LIN {X 0,Y 523.952,Z 123.214,A -85,B 0,C 180,E1 -4834.581,E2 -4834.581} C_VEL
LIN {X 0,Y 523.913,Z 123.226,A -85,B 0,C 180,E1 -4837.106,E2 -4837.106} C_VEL
LIN {X 0,Y 523.982,Z 123.211,A -85,B 0,C 180,E1 -4839.866,E2 -4839.866} C_VEL
LIN {X 0,Y 523.946,Z 123.22,A -85,B 0,C 180,E1 -4842.836,E2 -4842.836} C_VEL
LIN {X 0,Y 523.977,Z 123.217,A -85,B 0,C 180,E1 -4845.235,E2 -4845.235} C_VEL
LIN {X 0,Y 524.016,Z 123.21,A -85,B 0,C 180,E1 -4848.394,E2 -4848.394} C_VEL
LIN {X 0,Y 523.99,Z 123.212,A -85,B 0,C 180,E1 -4851.515,E2 -4851.515} C_VEL
LIN {X 0,Y 524.08,Z 123.208,A -85,B 0,C 180,E1 -4854.613,E2 -4854.613} C_VEL
LIN {X 0,Y 524.112,Z 123.197,A -85,B 0,C 180,E1 -4857.694,E2 -4857.694} C_VEL
LIN {X 0,Y 524.121,Z 123.2,A -85,B 0,C 180,E1 -4860.768,E2 -4860.768} C_VEL
LIN {X 0,Y 524.032,Z 123.209,A -85,B 0,C 180,E1 -4863.075,E2 -4863.075} C_VEL
LIN {X 0,Y 524.035,Z 123.213,A -85,B 0,C 180,E1 -4866.159,E2 -4866.159} C_VEL
LIN {X 0,Y 524.063,Z 123.317,A -85,B 0,C 180,E1 -4866.954,E2 -4866.954} C_VEL
LIN {X 0,Y 524.293,Z 129.392,A -85,B 0,C 180,E1 -4868.091,E2 -4868.091} C_VEL
LIN {X 0,Y 524.223,Z 139.02,A -85,B 0,C 180,E1 -4869.915,E2 -4869.915} C_VEL
LIN {X 0,Y 525.974,Z 147.912,A -85,B 0,C 180,E1 -4870.1,E2 -4870.1} C_VEL
LIN {X 0,Y 525.464,Z 245.35,A -85,B 0,C 180,E1 -4871.5,E2 -4871.5} C_VEL
LIN {X 0,Y 525.299,Z 258.517,A -85,B 0,C 180,E1 -4871.84,E2 -4871.84} C_VEL
LIN {X 0,Y 525.121,Z 270.833,A -85,B 0,C 180,E1 -4872.311,E2 -4872.311} C_VEL
LIN {X 0,Y 524.861,Z 283.293,A -85,B 0,C 180,E1 -4872.961,E2 -4872.961} C_VEL
LIN {X 0,Y 524.562,Z 295.002,A -85,B 0,C 180,E1 -4873.757,E2 -4873.757} C_VEL
LIN {X 0,Y 524.314,Z 305.505,A -85,B 0,C 180,E1 -4874.655,E2 -4874.655} C_VEL
LIN {X 0,Y 524.119,Z 314.056,A -85,B 0,C 180,E1 -4875.556,E2 -4875.556} C_VEL
LIN {X 0,Y 523.845,Z 323.352,A -85,B 0,C 180,E1 -4876.765,E2 -4876.765} C_VEL
LIN {X 0,Y 523.686,Z 330.798,A -85,B 0,C 180,E1 -4877.979,E2 -4877.979} C_VEL
LIN {X 0,Y 523.617,Z 336.668,A -85,B 0,C 180,E1 -4879.198,E2 -4879.198} C_VEL
LIN {X 0,Y 523.481,Z 341.276,A -85,B 0,C 180,E1 -4880.43,E2 -4880.43} C_VEL
LIN {X 0,Y 523.428,Z 343.689,A -85,B 0,C 180,E1 -4881.255,E2 -4881.255} C_VEL
LIN {X 0,Y 523.372,Z 345.621,A -85,B 0,C 180,E1 -4882.096,E2 -4882.096} C_VEL
LIN {X 0,Y 523.31,Z 347.024,A -85,B 0,C 180,E1 -4882.921,E2 -4882.921} C_VEL
LIN {X 0,Y 523.288,Z 348.184,A -85,B 0,C 180,E1 -4884.038,E2 -4884.038} C_VEL
LIN {X 0,Y 523.308,Z 348.449,A -85,B 0,C 180,E1 -4885.452,E2 -4885.452} C_VEL
LIN {X 0,Y 523.314,Z 347.985,A -85,B 0,C 180,E1 -4886.307,E2 -4886.307} C_VEL
LIN {X 0,Y 523.362,Z 346.319,A -85,B 0,C 180,E1 -4887.589,E2 -4887.589} C_VEL
LIN {X 0,Y 523.419,Z 343.417,A -85,B 0,C 180,E1 -4888.906,E2 -4888.906} C_VEL
LIN {X 0,Y 523.476,Z 339.204,A -85,B 0,C 180,E1 -4890.229,E2 -4890.229} C_VEL
LIN {X 0,Y 523.489,Z 338.508,A -85,B 0,C 180,E1 -4890.408,E2 -4890.408} C_VEL
LIN {X 0,Y 522.873,Z 336.184,A -85,B 0,C 180,E1 -4890.998,E2 -4890.998} C_VEL
LIN {X 0,Y 520.085,Z 331.973,A -85,B 0,C 180,E1 -4891.94,E2 -4891.94} C_VEL
LIN {X 0,Y 517.343,Z 327.2,A -85,B 0,C 180,E1 -4892.853,E2 -4892.853} C_VEL
LIN {X 0,Y 516.804,Z 323.835,A -85,B 0,C 180,E1 -4893.39,E2 -4893.39} C_VEL
LIN {X 0,Y 517.078,Z 314.887,A -85,B 0,C 180,E1 -4894.578,E2 -4894.578} C_VEL
LIN {X 0,Y 517.334,Z 305.085,A -85,B 0,C 180,E1 -4895.625,E2 -4895.625} C_VEL
LIN {X 0,Y 517.652,Z 294.078,A -85,B 0,C 180,E1 -4896.561,E2 -4896.561} C_VEL
LIN {X 0,Y 517.921,Z 283.602,A -85,B 0,C 180,E1 -4897.276,E2 -4897.276} C_VEL
LIN {X 0,Y 518.173,Z 272.168,A -85,B 0,C 180,E1 -4897.893,E2 -4897.893} C_VEL
LIN {X 0,Y 518.298,Z 259.428,A -85,B 0,C 180,E1 -4898.402,E2 -4898.402} C_VEL
LIN {X 0,Y 518.52,Z 246.192,A -85,B 0,C 180,E1 -4898.757,E2 -4898.757} C_VEL
LIN {X 0,Y 519.003,Z 147.832,A -85,B 0,C 180,E1 -4900.198,E2 -4900.198} C_VEL
LIN {X 0,Y 517.241,Z 138.787,A -85,B 0,C 180,E1 -4900.405,E2 -4900.405} C_VEL
LIN {X 0,Y 517.335,Z 126.807,A -85,B 0,C 180,E1 -4902.811,E2 -4902.811} C_VEL
LIN {X 0,Y 516.956,Z 124.094,A -85,B 0,C 180,E1 -4903.426,E2 -4903.426} C_VEL
LIN {X 0,Y 516.883,Z 124.101,A -85,B 0,C 180,E1 -4906.107,E2 -4906.107} C_VEL
LIN {X 0,Y 516.915,Z 124.092,A -85,B 0,C 180,E1 -4908.398,E2 -4908.398} C_VEL
LIN {X 0,Y 516.88,Z 124.099,A -85,B 0,C 180,E1 -4911.284,E2 -4911.284} C_VEL
LIN {X 0,Y 516.87,Z 124.098,A -85,B 0,C 180,E1 -4914.219,E2 -4914.219} C_VEL
LIN {X 0,Y 516.88,Z 124.098,A -85,B 0,C 180,E1 -4917.052,E2 -4917.052} C_VEL
LIN {X 0,Y 516.886,Z 124.098,A -85,B 0,C 180,E1 -4919.796,E2 -4919.796} C_VEL
LIN {X 0,Y 516.925,Z 124.089,A -85,B 0,C 180,E1 -4922.467,E2 -4922.467} C_VEL
LIN {X 0,Y 516.908,Z 124.096,A -85,B 0,C 180,E1 -4925.071,E2 -4925.071} C_VEL
LIN {X 0,Y 516.885,Z 124.095,A -85,B 0,C 180,E1 -4928.462,E2 -4928.462} C_VEL
LIN {X 0,Y 516.899,Z 124.098,A -85,B 0,C 180,E1 -4930.954,E2 -4930.954} C_VEL
LIN {X 0,Y 516.907,Z 124.097,A -85,B 0,C 180,E1 -4933.41,E2 -4933.41} C_VEL
LIN {X 0,Y 516.894,Z 124.094,A -85,B 0,C 180,E1 -4935.833,E2 -4935.833} C_VEL
LIN {X 0,Y 516.965,Z 124.085,A -85,B 0,C 180,E1 -4938.233,E2 -4938.233} C_VEL
LIN {X 0,Y 516.967,Z 124.088,A -85,B 0,C 180,E1 -4941.399,E2 -4941.399} C_VEL
LIN {X 0,Y 517.001,Z 124.08,A -85,B 0,C 180,E1 -4943.756,E2 -4943.756} C_VEL
LIN {X 0,Y 517.012,Z 124.088,A -85,B 0,C 180,E1 -4946.883,E2 -4946.883} C_VEL
LIN {X 0,Y 517.085,Z 124.07,A -85,B 0,C 180,E1 -4950,E2 -4950} C_VEL
LIN {X 0,Y 517.01,Z 124.083,A -85,B 0,C 180,E1 -4953.117,E2 -4953.117} C_VEL
LIN {X 0,Y 517.002,Z 124.083,A -85,B 0,C 180,E1 -4956.243,E2 -4956.243} C_VEL
LIN {X 0,Y 516.952,Z 124.087,A -85,B 0,C 180,E1 -4959.389,E2 -4959.389} C_VEL
LIN {X 0,Y 516.951,Z 124.087,A -85,B 0,C 180,E1 -4961.807,E2 -4961.807} C_VEL
LIN {X 0,Y 516.945,Z 124.088,A -85,B 0,C 180,E1 -4965.147,E2 -4965.147} C_VEL
LIN {X 0,Y 516.923,Z 124.096,A -85,B 0,C 180,E1 -4968.222,E2 -4968.222} C_VEL
LIN {X 0,Y 516.91,Z 124.095,A -85,B 0,C 180,E1 -4970.701,E2 -4970.701} C_VEL
LIN {X 0,Y 516.888,Z 124.1,A -85,B 0,C 180,E1 -4974.073,E2 -4974.073} C_VEL
LIN {X 0,Y 516.922,Z 124.093,A -85,B 0,C 180,E1 -4976.658,E2 -4976.658} C_VEL
LIN {X 0,Y 516.917,Z 124.092,A -85,B 0,C 180,E1 -4979.525,E2 -4979.525} C_VEL
LIN {X 0,Y 516.898,Z 124.096,A -85,B 0,C 180,E1 -4982.544,E2 -4982.544} C_VEL
LIN {X 0,Y 516.877,Z 124.096,A -85,B 0,C 180,E1 -4985.332,E2 -4985.332} C_VEL
LIN {X 0,Y 516.879,Z 124.104,A -85,B 0,C 180,E1 -4987.943,E2 -4987.943} C_VEL
LIN {X 0,Y 516.883,Z 124.095,A -85,B 0,C 180,E1 -4990.741,E2 -4990.741} C_VEL
LIN {X 0,Y 516.902,Z 124.092,A -85,B 0,C 180,E1 -4992.829,E2 -4992.829} C_VEL
LIN {X 0,Y 516.919,Z 124.09,A -85,B 0,C 180,E1 -4995.01,E2 -4995.01} C_VEL
LIN {X 0,Y 516.92,Z 124.091,A -85,B 0,C 180,E1 -4998.398,E2 -4998.398} C_VEL
LIN {X 0,Y 516.884,Z 124.098,A -85,B 0,C 180,E1 -5001.285,E2 -5001.285} C_VEL
LIN {X 0,Y 516.868,Z 124.098,A -85,B 0,C 180,E1 -5004.22,E2 -5004.22} C_VEL
LIN {X 0,Y 516.894,Z 124.095,A -85,B 0,C 180,E1 -5007.053,E2 -5007.053} C_VEL
LIN {X 0,Y 516.889,Z 124.099,A -85,B 0,C 180,E1 -5009.796,E2 -5009.796} C_VEL
LIN {X 0,Y 516.925,Z 124.089,A -85,B 0,C 180,E1 -5012.468,E2 -5012.468} C_VEL
LIN {X 0,Y 516.906,Z 124.096,A -85,B 0,C 180,E1 -5015.072,E2 -5015.072} C_VEL
LIN {X 0,Y 516.883,Z 124.095,A -85,B 0,C 180,E1 -5018.462,E2 -5018.462} C_VEL
LIN {X 0,Y 516.901,Z 124.097,A -85,B 0,C 180,E1 -5020.955,E2 -5020.955} C_VEL
LIN {X 0,Y 516.911,Z 124.098,A -85,B 0,C 180,E1 -5023.41,E2 -5023.41} C_VEL
LIN {X 0,Y 516.892,Z 124.095,A -85,B 0,C 180,E1 -5025.834,E2 -5025.834} C_VEL
LIN {X 0,Y 516.963,Z 124.085,A -85,B 0,C 180,E1 -5028.234,E2 -5028.234} C_VEL
LIN {X 0,Y 516.966,Z 124.088,A -85,B 0,C 180,E1 -5031.4,E2 -5031.4} C_VEL
LIN {X 0,Y 517.001,Z 124.081,A -85,B 0,C 180,E1 -5033.757,E2 -5033.757} C_VEL
LIN {X 0,Y 517.011,Z 124.087,A -85,B 0,C 180,E1 -5036.883,E2 -5036.883} C_VEL
LIN {X 0,Y 517.084,Z 124.07,A -85,B 0,C 180,E1 -5040,E2 -5040} C_VEL
LIN {X 0,Y 517.01,Z 124.083,A -85,B 0,C 180,E1 -5043.117,E2 -5043.117} C_VEL
LIN {X 0,Y 517.014,Z 124.081,A -85,B 0,C 180,E1 -5046.243,E2 -5046.243} C_VEL
LIN {X 0,Y 516.953,Z 124.087,A -85,B 0,C 180,E1 -5049.39,E2 -5049.39} C_VEL
LIN {X 0,Y 516.951,Z 124.087,A -85,B 0,C 180,E1 -5051.808,E2 -5051.808} C_VEL
LIN {X 0,Y 516.946,Z 124.088,A -85,B 0,C 180,E1 -5055.148,E2 -5055.148} C_VEL
LIN {X 0,Y 516.924,Z 124.095,A -85,B 0,C 180,E1 -5058.223,E2 -5058.223} C_VEL
LIN {X 0,Y 516.912,Z 124.096,A -85,B 0,C 180,E1 -5060.702,E2 -5060.702} C_VEL
LIN {X 0,Y 516.89,Z 124.099,A -85,B 0,C 180,E1 -5064.073,E2 -5064.073} C_VEL
LIN {X 0,Y 516.924,Z 124.093,A -85,B 0,C 180,E1 -5066.658,E2 -5066.658} C_VEL
LIN {X 0,Y 516.91,Z 124.092,A -85,B 0,C 180,E1 -5069.524,E2 -5069.524} C_VEL
LIN {X 0,Y 516.895,Z 124.097,A -85,B 0,C 180,E1 -5072.544,E2 -5072.544} C_VEL
LIN {X 0,Y 516.865,Z 124.097,A -85,B 0,C 180,E1 -5075.33,E2 -5075.33} C_VEL
LIN {X 0,Y 516.881,Z 124.102,A -85,B 0,C 180,E1 -5077.944,E2 -5077.944} C_VEL
LIN {X 0,Y 516.895,Z 124.094,A -85,B 0,C 180,E1 -5080.741,E2 -5080.741} C_VEL
LIN {X 0,Y 516.883,Z 124.104,A -85,B 0,C 180,E1 -5083.904,E2 -5083.904} C_VEL
LIN {X 0,Y 516.883,Z 124.1,A -85,B 0,C 180,E1 -5086.107,E2 -5086.107} C_VEL
LIN {X 0,Y 516.917,Z 124.092,A -85,B 0,C 180,E1 -5088.399,E2 -5088.399} C_VEL
LIN {X 0,Y 516.884,Z 124.097,A -85,B 0,C 180,E1 -5091.285,E2 -5091.285} C_VEL
LIN {X 0,Y 516.872,Z 124.098,A -85,B 0,C 180,E1 -5094.22,E2 -5094.22} C_VEL
LIN {X 0,Y 516.896,Z 124.095,A -85,B 0,C 180,E1 -5097.053,E2 -5097.053} C_VEL
LIN {X 0,Y 516.893,Z 124.1,A -85,B 0,C 180,E1 -5099.797,E2 -5099.797} C_VEL
LIN {X 0,Y 516.928,Z 124.091,A -85,B 0,C 180,E1 -5102.468,E2 -5102.468} C_VEL
LIN {X 0,Y 516.957,Z 124.191,A -85,B 0,C 180,E1 -5104.402,E2 -5104.402} C_VEL
LIN {X 0,Y 518.636,Z 133.005,A -85,B 0,C 180,E1 -5105.836,E2 -5105.836} C_VEL
LIN {X 0,Y 518.274,Z 148.017,A -85,B 0,C 180,E1 -5108.105,E2 -5108.105} C_VEL
LIN {X 0,Y 517.818,Z 167.379,A -85,B 0,C 180,E1 -5110.99,E2 -5110.99} C_VEL
LIN {X 0,Y 517.345,Z 186.704,A -85,B 0,C 180,E1 -5113.83,E2 -5113.83} C_VEL
LIN {X 0,Y 517.246,Z 192.193,A -85,B 0,C 180,E1 -5114.633,E2 -5114.633} C_VEL
LIN {X 0,Y 518.989,Z 205.615,A -85,B 0,C 180,E1 -5114.884,E2 -5114.884} C_VEL
LIN {X 0,Y 518.489,Z 301.678,A -85,B 0,C 180,E1 -5116.278,E2 -5116.278} C_VEL
LIN {X 0,Y 518.244,Z 314.629,A -85,B 0,C 180,E1 -5116.622,E2 -5116.622} C_VEL
LIN {X 0,Y 517.964,Z 327.229,A -85,B 0,C 180,E1 -5117.113,E2 -5117.113} C_VEL
LIN {X 0,Y 517.645,Z 339.245,A -85,B 0,C 180,E1 -5117.752,E2 -5117.752} C_VEL
LIN {X 0,Y 517.35,Z 350.788,A -85,B 0,C 180,E1 -5118.541,E2 -5118.541} C_VEL
LIN {X 0,Y 517.118,Z 361.192,A -85,B 0,C 180,E1 -5119.428,E2 -5119.428} C_VEL
LIN {X 0,Y 516.831,Z 370.527,A -85,B 0,C 180,E1 -5120.411,E2 -5120.411} C_VEL
LIN {X 0,Y 516.617,Z 379.595,A -85,B 0,C 180,E1 -5121.591,E2 -5121.591} C_VEL
LIN {X 0,Y 516.461,Z 386.898,A -85,B 0,C 180,E1 -5122.769,E2 -5122.769} C_VEL
LIN {X 0,Y 516.372,Z 391.826,A -85,B 0,C 180,E1 -5123.749,E2 -5123.749} C_VEL
LIN {X 0,Y 516.312,Z 396.613,A -85,B 0,C 180,E1 -5124.924,E2 -5124.924} C_VEL
LIN {X 0,Y 516.37,Z 400.275,A -85,B 0,C 180,E1 -5126.098,E2 -5126.098} C_VEL
LIN {X 0,Y 516.327,Z 402.159,A -85,B 0,C 180,E1 -5126.879,E2 -5126.879} C_VEL
LIN {X 0,Y 516.266,Z 403.569,A -85,B 0,C 180,E1 -5127.66,E2 -5127.66} C_VEL
LIN {X 0,Y 516.182,Z 405.179,A -85,B 0,C 180,E1 -5129.22,E2 -5129.22} C_VEL
LIN {X 0,Y 516.186,Z 405.391,A -85,B 0,C 180,E1 -5130,E2 -5130} C_VEL
LIN {X 0,Y 516.182,Z 405.165,A -85,B 0,C 180,E1 -5130.78,E2 -5130.78} C_VEL
LIN {X 0,Y 516.266,Z 403.524,A -85,B 0,C 180,E1 -5132.341,E2 -5132.341} C_VEL
LIN {X 0,Y 516.327,Z 402.097,A -85,B 0,C 180,E1 -5133.121,E2 -5133.121} C_VEL
LIN {X 0,Y 516.312,Z 399.099,A -85,B 0,C 180,E1 -5134.294,E2 -5134.294} C_VEL
LIN {X 0,Y 516.389,Z 395.048,A -85,B 0,C 180,E1 -5135.467,E2 -5135.467} C_VEL
LIN {X 0,Y 516.416,Z 388.803,A -85,B 0,C 180,E1 -5136.84,E2 -5136.84} C_VEL
LIN {X 0,Y 516.563,Z 381.996,A -85,B 0,C 180,E1 -5138.017,E2 -5138.017} C_VEL
LIN {X 0,Y 516.74,Z 373.54,A -85,B 0,C 180,E1 -5139.196,E2 -5139.196} C_VEL
LIN {X 0,Y 516.935,Z 364.836,A -85,B 0,C 180,E1 -5140.18,E2 -5140.18} C_VEL
LIN {X 0,Y 517.253,Z 354.109,A -85,B 0,C 180,E1 -5141.164,E2 -5141.164} C_VEL
LIN {X 0,Y 517.492,Z 342.601,A -85,B 0,C 180,E1 -5142.012,E2 -5142.012} C_VEL
LIN {X 0,Y 517.793,Z 330.687,A -85,B 0,C 180,E1 -5142.692,E2 -5142.692} C_VEL
LIN {X 0,Y 518.108,Z 318.162,A -85,B 0,C 180,E1 -5143.233,E2 -5143.233} C_VEL
LIN {X 0,Y 518.355,Z 305.212,A -85,B 0,C 180,E1 -5143.626,E2 -5143.626} C_VEL
LIN {X 0,Y 518.548,Z 289.822,A -85,B 0,C 180,E1 -5143.895,E2 -5143.895} C_VEL
LIN {X 0,Y 518.851,Z 203.924,A -85,B 0,C 180,E1 -5145.135,E2 -5145.135} C_VEL
LIN {X 0,Y 517.179,Z 191.339,A -85,B 0,C 180,E1 -5145.382,E2 -5145.382} C_VEL
LIN {X 0,Y 517.63,Z 168.939,A -85,B 0,C 180,E1 -5148.607,E2 -5148.607} C_VEL
LIN {X 0,Y 517.938,Z 149.08,A -85,B 0,C 180,E1 -5151.492,E2 -5151.492} C_VEL
LIN {X 0,Y 518.301,Z 132.004,A -85,B 0,C 180,E1 -5154.004,E2 -5154.004} C_VEL
LIN {X 0,Y 516.973,Z 124.09,A -85,B 0,C 180,E1 -5155.248,E2 -5155.248} C_VEL
LIN {X 0,Y 516.922,Z 124.102,A -85,B 0,C 180,E1 -5158.415,E2 -5158.415} C_VEL
LIN {X 0,Y 516.893,Z 124.098,A -85,B 0,C 180,E1 -5161.11,E2 -5161.11} C_VEL
LIN {X 0,Y 516.912,Z 124.098,A -85,B 0,C 180,E1 -5163.966,E2 -5163.966} C_VEL
LIN {X 0,Y 516.88,Z 124.098,A -85,B 0,C 180,E1 -5166.746,E2 -5166.746} C_VEL
LIN {X 0,Y 516.886,Z 124.101,A -85,B 0,C 180,E1 -5169.721,E2 -5169.721} C_VEL
LIN {X 0,Y 516.915,Z 124.098,A -85,B 0,C 180,E1 -5171.775,E2 -5171.775} C_VEL
LIN {X 0,Y 516.927,Z 124.091,A -85,B 0,C 180,E1 -5175.01,E2 -5175.01} C_VEL
LIN {X 0,Y 516.917,Z 124.091,A -85,B 0,C 180,E1 -5178.399,E2 -5178.399} C_VEL
LIN {X 0,Y 516.884,Z 124.097,A -85,B 0,C 180,E1 -5181.284,E2 -5181.284} C_VEL
LIN {X 0,Y 516.874,Z 124.097,A -85,B 0,C 180,E1 -5184.22,E2 -5184.22} C_VEL
LIN {X 0,Y 516.884,Z 124.096,A -85,B 0,C 180,E1 -5187.052,E2 -5187.052} C_VEL
LIN {X 0,Y 516.89,Z 124.098,A -85,B 0,C 180,E1 -5189.796,E2 -5189.796} C_VEL
LIN {X 0,Y 516.928,Z 124.09,A -85,B 0,C 180,E1 -5192.467,E2 -5192.467} C_VEL
LIN {X 0,Y 516.909,Z 124.096,A -85,B 0,C 180,E1 -5195.071,E2 -5195.071} C_VEL
LIN {X 0,Y 516.888,Z 124.096,A -85,B 0,C 180,E1 -5198.462,E2 -5198.462} C_VEL
LIN {X 0,Y 516.895,Z 124.1,A -85,B 0,C 180,E1 -5200.954,E2 -5200.954} C_VEL
LIN {X 0,Y 516.901,Z 124.096,A -85,B 0,C 180,E1 -5203.409,E2 -5203.409} C_VEL
LIN {X 0,Y 516.89,Z 124.095,A -85,B 0,C 180,E1 -5205.833,E2 -5205.833} C_VEL
LIN {X 0,Y 516.953,Z 124.094,A -85,B 0,C 180,E1 -5209.028,E2 -5209.028} C_VEL
LIN {X 0,Y 516.965,Z 124.089,A -85,B 0,C 180,E1 -5212.186,E2 -5212.186} C_VEL
LIN {X 0,Y 517.027,Z 124.086,A -85,B 0,C 180,E1 -5214.54,E2 -5214.54} C_VEL
LIN {X 0,Y 517.083,Z 124.073,A -85,B 0,C 180,E1 -5217.663,E2 -5217.663} C_VEL
LIN {X 0,Y 517.091,Z 124.076,A -85,B 0,C 180,E1 -5220.778,E2 -5220.778} C_VEL
LIN {X 0,Y 516.974,Z 124.088,A -85,B 0,C 180,E1 -5223.117,E2 -5223.117} C_VEL
LIN {X 0,Y 517.001,Z 124.09,A -85,B 0,C 180,E1 -5226.243,E2 -5226.243} C_VEL
LIN {X 0,Y 516.988,Z 124.135,A -85,B 0,C 180,E1 -5226.817,E2 -5226.817} C_VEL
LIN {X 0,Y 517.351,Z 129.359,A -85,B 0,C 180,E1 -5227.807,E2 -5227.807} C_VEL
LIN {X 0,Y 517.256,Z 139.386,A -85,B 0,C 180,E1 -5229.704,E2 -5229.704} C_VEL
LIN {X 0,Y 519.133,Z 149.215,A -85,B 0,C 180,E1 -5229.915,E2 -5229.915} C_VEL
LIN {X 0,Y 518.556,Z 246.037,A -85,B 0,C 180,E1 -5231.333,E2 -5231.333} C_VEL
LIN {X 0,Y 518.384,Z 259.286,A -85,B 0,C 180,E1 -5231.684,E2 -5231.684} C_VEL
LIN {X 0,Y 518.205,Z 272.025,A -85,B 0,C 180,E1 -5232.185,E2 -5232.185} C_VEL
LIN {X 0,Y 517.906,Z 284.191,A -85,B 0,C 180,E1 -5232.839,E2 -5232.839} C_VEL
LIN {X 0,Y 517.6,Z 295.81,A -85,B 0,C 180,E1 -5233.645,E2 -5233.645} C_VEL
LIN {X 0,Y 517.311,Z 306.237,A -85,B 0,C 180,E1 -5234.556,E2 -5234.556} C_VEL
LIN {X 0,Y 517.063,Z 315.866,A -85,B 0,C 180,E1 -5235.607,E2 -5235.607} C_VEL
LIN {X 0,Y 516.81,Z 324.684,A -85,B 0,C 180,E1 -5236.796,E2 -5236.796} C_VEL
LIN {X 0,Y 516.638,Z 331.539,A -85,B 0,C 180,E1 -5237.956,E2 -5237.956} C_VEL
LIN {X 0,Y 516.552,Z 336.797,A -85,B 0,C 180,E1 -5239.058,E2 -5239.058} C_VEL
LIN {X 0,Y 516.431,Z 340.847,A -85,B 0,C 180,E1 -5240.114,E2 -5240.114} C_VEL
LIN {X 0,Y 516.331,Z 344.945,A -85,B 0,C 180,E1 -5241.562,E2 -5241.562} C_VEL
LIN {X 0,Y 516.262,Z 346.658,A -85,B 0,C 180,E1 -5242.406,E2 -5242.406} C_VEL
LIN {X 0,Y 516.205,Z 347.893,A -85,B 0,C 180,E1 -5243.255,E2 -5243.255} C_VEL
LIN {X 0,Y 516.19,Z 348.67,A -85,B 0,C 180,E1 -5244.186,E2 -5244.186} C_VEL
LIN {X 0,Y 516.185,Z 348.913,A -85,B 0,C 180,E1 -5244.965,E2 -5244.965} C_VEL
LIN {X 0,Y 516.248,Z 348.561,A -85,B 0,C 180,E1 -5246.038,E2 -5246.038} C_VEL
LIN {X 0,Y 516.274,Z 346.801,A -85,B 0,C 180,E1 -5247.57,E2 -5247.57} C_VEL
LIN {X 0,Y 516.334,Z 343.965,A -85,B 0,C 180,E1 -5248.894,E2 -5248.894} C_VEL
LIN {X 0,Y 516.406,Z 339.798,A -85,B 0,C 180,E1 -5250.235,E2 -5250.235} C_VEL
LIN {X 0,Y 516.577,Z 334.142,A -85,B 0,C 180,E1 -5251.586,E2 -5251.586} C_VEL
LIN {X 0,Y 516.746,Z 328.229,A -85,B 0,C 180,E1 -5252.696,E2 -5252.696} C_VEL
LIN {X 0,Y 516.804,Z 323.835,A -85,B 0,C 180,E1 -5253.39,E2 -5253.39} C_VEL
LIN {X 0,Y 516.268,Z 320.293,A -85,B 0,C 180,E1 -5253.912,E2 -5253.912} C_VEL
LIN {X 0,Y 513.569,Z 314.279,A -85,B 0,C 180,E1 -5254.739,E2 -5254.739} C_VEL
LIN {X 0,Y 510.892,Z 307.742,A -85,B 0,C 180,E1 -5255.518,E2 -5255.518} C_VEL
LIN {X 0,Y 510.388,Z 303.34,A -85,B 0,C 180,E1 -5255.958,E2 -5255.958} C_VEL
LIN {X 0,Y 510.733,Z 292.231,A -85,B 0,C 180,E1 -5256.879,E2 -5256.879} C_VEL
LIN {X 0,Y 511.009,Z 281.019,A -85,B 0,C 180,E1 -5257.611,E2 -5257.611} C_VEL
LIN {X 0,Y 511.278,Z 269.154,A -85,B 0,C 180,E1 -5258.211,E2 -5258.211} C_VEL
LIN {X 0,Y 511.487,Z 256.568,A -85,B 0,C 180,E1 -5258.68,E2 -5258.68} C_VEL
LIN {X 0,Y 511.678,Z 243.597,A -85,B 0,C 180,E1 -5258.992,E2 -5258.992} C_VEL
LIN {X 0,Y 512.209,Z 149.22,A -85,B 0,C 180,E1 -5260.382,E2 -5260.382} C_VEL
LIN {X 0,Y 510.234,Z 139.088,A -85,B 0,C 180,E1 -5260.617,E2 -5260.617} C_VEL
LIN {X 0,Y 510.362,Z 128.466,A -85,B 0,C 180,E1 -5262.765,E2 -5262.765} C_VEL
LIN {X 0,Y 509.924,Z 124.97,A -85,B 0,C 180,E1 -5263.524,E2 -5263.524} C_VEL
LIN {X 0,Y 509.82,Z 124.978,A -85,B 0,C 180,E1 -5266.428,E2 -5266.428} C_VEL
LIN {X 0,Y 509.839,Z 124.976,A -85,B 0,C 180,E1 -5269.302,E2 -5269.302} C_VEL
LIN {X 0,Y 509.851,Z 124.977,A -85,B 0,C 180,E1 -5271.786,E2 -5271.786} C_VEL
LIN {X 0,Y 509.829,Z 124.973,A -85,B 0,C 180,E1 -5274.622,E2 -5274.622} C_VEL
LIN {X 0,Y 509.859,Z 124.978,A -85,B 0,C 180,E1 -5277.48,E2 -5277.48} C_VEL
LIN {X 0,Y 509.857,Z 124.97,A -85,B 0,C 180,E1 -5280.273,E2 -5280.273} C_VEL
LIN {X 0,Y 509.883,Z 124.97,A -85,B 0,C 180,E1 -5282.944,E2 -5282.944} C_VEL
LIN {X 0,Y 509.864,Z 124.975,A -85,B 0,C 180,E1 -5285.573,E2 -5285.573} C_VEL
LIN {X 0,Y 509.849,Z 124.976,A -85,B 0,C 180,E1 -5288.998,E2 -5288.998} C_VEL
LIN {X 0,Y 509.86,Z 124.974,A -85,B 0,C 180,E1 -5291.516,E2 -5291.516} C_VEL
LIN {X 0,Y 509.852,Z 124.971,A -85,B 0,C 180,E1 -5293.997,E2 -5293.997} C_VEL
LIN {X 0,Y 509.861,Z 124.97,A -85,B 0,C 180,E1 -5296.448,E2 -5296.448} C_VEL
LIN {X 0,Y 509.913,Z 124.969,A -85,B 0,C 180,E1 -5298.874,E2 -5298.874} C_VEL
LIN {X 0,Y 509.951,Z 124.958,A -85,B 0,C 180,E1 -5302.078,E2 -5302.078} C_VEL
LIN {X 0,Y 509.978,Z 124.957,A -85,B 0,C 180,E1 -5304.464,E2 -5304.464} C_VEL
LIN {X 0,Y 510.055,Z 124.946,A -85,B 0,C 180,E1 -5307.631,E2 -5307.631} C_VEL
LIN {X 0,Y 510.063,Z 124.953,A -85,B 0,C 180,E1 -5310.789,E2 -5310.789} C_VEL
LIN {X 0,Y 509.952,Z 124.961,A -85,B 0,C 180,E1 -5313.16,E2 -5313.16} C_VEL
LIN {X 0,Y 509.953,Z 124.962,A -85,B 0,C 180,E1 -5316.33,E2 -5316.33} C_VEL
LIN {X 0,Y 509.914,Z 124.97,A -85,B 0,C 180,E1 -5318.72,E2 -5318.72} C_VEL
LIN {X 0,Y 509.903,Z 124.966,A -85,B 0,C 180,E1 -5321.931,E2 -5321.931} C_VEL
LIN {X 0,Y 509.892,Z 124.966,A -85,B 0,C 180,E1 -5325.242,E2 -5325.242} C_VEL
LIN {X 0,Y 509.886,Z 124.969,A -85,B 0,C 180,E1 -5328.001,E2 -5328.001} C_VEL
LIN {X 0,Y 509.848,Z 124.972,A -85,B 0,C 180,E1 -5331.001,E2 -5331.001} C_VEL
LIN {X 0,Y 509.82,Z 124.975,A -85,B 0,C 180,E1 -5333.564,E2 -5333.564} C_VEL
LIN {X 0,Y 509.908,Z 124.97,A -85,B 0,C 180,E1 -5336.378,E2 -5336.378} C_VEL
LIN {X 0,Y 509.878,Z 124.968,A -85,B 0,C 180,E1 -5338.844,E2 -5338.844} C_VEL
LIN {X 0,Y 509.824,Z 124.976,A -85,B 0,C 180,E1 -5341.589,E2 -5341.589} C_VEL
LIN {X 0,Y 509.849,Z 124.975,A -85,B 0,C 180,E1 -5344.413,E2 -5344.413} C_VEL
LIN {X 0,Y 509.816,Z 124.976,A -85,B 0,C 180,E1 -5347.34,E2 -5347.34} C_VEL
LIN {X 0,Y 509.836,Z 124.976,A -85,B 0,C 180,E1 -5350.382,E2 -5350.382} C_VEL
LIN {X 0,Y 509.836,Z 124.973,A -85,B 0,C 180,E1 -5353.064,E2 -5353.064} C_VEL
LIN {X 0,Y 509.828,Z 124.982,A -85,B 0,C 180,E1 -5355.792,E2 -5355.792} C_VEL
LIN {X 0,Y 509.862,Z 124.97,A -85,B 0,C 180,E1 -5358.576,E2 -5358.576} C_VEL
LIN {X 0,Y 509.849,Z 124.979,A -85,B 0,C 180,E1 -5361.786,E2 -5361.786} C_VEL
LIN {X 0,Y 509.826,Z 124.974,A -85,B 0,C 180,E1 -5364.622,E2 -5364.622} C_VEL
LIN {X 0,Y 509.863,Z 124.977,A -85,B 0,C 180,E1 -5367.481,E2 -5367.481} C_VEL
LIN {X 0,Y 509.855,Z 124.971,A -85,B 0,C 180,E1 -5370.274,E2 -5370.274} C_VEL
LIN {X 0,Y 509.882,Z 124.969,A -85,B 0,C 180,E1 -5372.945,E2 -5372.945} C_VEL
LIN {X 0,Y 509.862,Z 124.976,A -85,B 0,C 180,E1 -5375.574,E2 -5375.574} C_VEL
LIN {X 0,Y 509.848,Z 124.975,A -85,B 0,C 180,E1 -5378.999,E2 -5378.999} C_VEL
LIN {X 0,Y 509.886,Z 124.967,A -85,B 0,C 180,E1 -5381.999,E2 -5381.999} C_VEL
LIN {X 0,Y 509.908,Z 124.967,A -85,B 0,C 180,E1 -5384.819,E2 -5384.819} C_VEL
LIN {X 0,Y 509.899,Z 124.965,A -85,B 0,C 180,E1 -5388.124,E2 -5388.124} C_VEL
LIN {X 0,Y 509.913,Z 124.969,A -85,B 0,C 180,E1 -5391.28,E2 -5391.28} C_VEL
LIN {X 0,Y 509.952,Z 124.959,A -85,B 0,C 180,E1 -5393.67,E2 -5393.67} C_VEL
LIN {X 0,Y 509.953,Z 124.965,A -85,B 0,C 180,E1 -5396.84,E2 -5396.84} C_VEL
LIN {X 0,Y 510.061,Z 124.949,A -85,B 0,C 180,E1 -5399.211,E2 -5399.211} C_VEL
LIN {X 0,Y 510.055,Z 124.948,A -85,B 0,C 180,E1 -5402.369,E2 -5402.369} C_VEL
LIN {X 0,Y 509.981,Z 124.958,A -85,B 0,C 180,E1 -5406.33,E2 -5406.33} C_VEL
LIN {X 0,Y 509.915,Z 124.971,A -85,B 0,C 180,E1 -5408.721,E2 -5408.721} C_VEL
LIN {X 0,Y 509.903,Z 124.965,A -85,B 0,C 180,E1 -5411.932,E2 -5411.932} C_VEL
LIN {X 0,Y 509.893,Z 124.966,A -85,B 0,C 180,E1 -5415.242,E2 -5415.242} C_VEL
LIN {X 0,Y 509.888,Z 124.969,A -85,B 0,C 180,E1 -5418.001,E2 -5418.001} C_VEL
LIN {X 0,Y 509.849,Z 124.973,A -85,B 0,C 180,E1 -5421.002,E2 -5421.002} C_VEL
LIN {X 0,Y 509.821,Z 124.975,A -85,B 0,C 180,E1 -5423.564,E2 -5423.564} C_VEL
LIN {X 0,Y 509.91,Z 124.971,A -85,B 0,C 180,E1 -5426.379,E2 -5426.379} C_VEL
LIN {X 0,Y 509.875,Z 124.969,A -85,B 0,C 180,E1 -5428.845,E2 -5428.845} C_VEL
LIN {X 0,Y 509.819,Z 124.976,A -85,B 0,C 180,E1 -5431.591,E2 -5431.591} C_VEL
LIN {X 0,Y 509.847,Z 124.976,A -85,B 0,C 180,E1 -5434.414,E2 -5434.414} C_VEL
LIN {X 0,Y 509.817,Z 124.976,A -85,B 0,C 180,E1 -5437.341,E2 -5437.341} C_VEL
LIN {X 0,Y 509.858,Z 124.973,A -85,B 0,C 180,E1 -5440.381,E2 -5440.381} C_VEL
LIN {X 0,Y 509.824,Z 124.974,A -85,B 0,C 180,E1 -5443.063,E2 -5443.063} C_VEL
LIN {X 0,Y 509.832,Z 124.981,A -85,B 0,C 180,E1 -5445.793,E2 -5445.793} C_VEL
LIN {X 0,Y 509.859,Z 124.97,A -85,B 0,C 180,E1 -5448.575,E2 -5448.575} C_VEL
LIN {X 0,Y 509.852,Z 124.979,A -85,B 0,C 180,E1 -5451.787,E2 -5451.787} C_VEL
LIN {X 0,Y 509.831,Z 124.973,A -85,B 0,C 180,E1 -5454.622,E2 -5454.622} C_VEL
LIN {X 0,Y 509.862,Z 124.976,A -85,B 0,C 180,E1 -5457.481,E2 -5457.481} C_VEL
LIN {X 0,Y 509.86,Z 124.971,A -85,B 0,C 180,E1 -5460.274,E2 -5460.274} C_VEL
LIN {X 0,Y 509.885,Z 124.971,A -85,B 0,C 180,E1 -5462.945,E2 -5462.945} C_VEL
LIN {X 0,Y 509.937,Z 125.056,A -85,B 0,C 180,E1 -5464.215,E2 -5464.215} C_VEL
LIN {X 0,Y 511.732,Z 135.217,A -85,B 0,C 180,E1 -5465.885,E2 -5465.885} C_VEL
LIN {X 0,Y 511.174,Z 155.976,A -85,B 0,C 180,E1 -5469.056,E2 -5469.056} C_VEL
LIN {X 0,Y 510.59,Z 178.078,A -85,B 0,C 180,E1 -5472.373,E2 -5472.373} C_VEL
LIN {X 0,Y 510.242,Z 191.99,A -85,B 0,C 180,E1 -5474.42,E2 -5474.42} C_VEL
LIN {X 0,Y 512.12,Z 206.484,A -85,B 0,C 180,E1 -5474.694,E2 -5474.694} C_VEL
LIN {X 0,Y 511.585,Z 300.889,A -85,B 0,C 180,E1 -5476.09,E2 -5476.09} C_VEL
LIN {X 0,Y 511.338,Z 313.21,A -85,B 0,C 180,E1 -5476.412,E2 -5476.412} C_VEL
LIN {X 0,Y 511.053,Z 325.511,A -85,B 0,C 180,E1 -5476.885,E2 -5476.885} C_VEL
LIN {X 0,Y 510.729,Z 336.846,A -85,B 0,C 180,E1 -5477.469,E2 -5477.469} C_VEL
LIN {X 0,Y 510.396,Z 347.685,A -85,B 0,C 180,E1 -5478.181,E2 -5478.181} C_VEL
LIN {X 0,Y 510.165,Z 358.562,A -85,B 0,C 180,E1 -5479.081,E2 -5479.081} C_VEL
LIN {X 0,Y 509.811,Z 368.343,A -85,B 0,C 180,E1 -5480.078,E2 -5480.078} C_VEL
LIN {X 0,Y 509.625,Z 376.37,A -85,B 0,C 180,E1 -5481.075,E2 -5481.075} C_VEL
LIN {X 0,Y 509.427,Z 384.218,A -85,B 0,C 180,E1 -5482.27,E2 -5482.27} C_VEL
LIN {X 0,Y 509.288,Z 391.419,A -85,B 0,C 180,E1 -5483.662,E2 -5483.662} C_VEL
LIN {X 0,Y 509.244,Z 396.216,A -85,B 0,C 180,E1 -5484.854,E2 -5484.854} C_VEL
LIN {X 0,Y 509.275,Z 399.882,A -85,B 0,C 180,E1 -5486.044,E2 -5486.044} C_VEL
LIN {X 0,Y 509.241,Z 401.77,A -85,B 0,C 180,E1 -5486.836,E2 -5486.836} C_VEL
LIN {X 0,Y 509.196,Z 403.184,A -85,B 0,C 180,E1 -5487.627,E2 -5487.627} C_VEL
LIN {X 0,Y 509.094,Z 404.792,A -85,B 0,C 180,E1 -5489.209,E2 -5489.209} C_VEL
LIN {X 0,Y 509.097,Z 405.004,A -85,B 0,C 180,E1 -5490,E2 -5490} C_VEL
LIN {X 0,Y 509.094,Z 404.776,A -85,B 0,C 180,E1 -5490.791,E2 -5490.791} C_VEL
LIN {X 0,Y 509.196,Z 403.127,A -85,B 0,C 180,E1 -5492.373,E2 -5492.373} C_VEL
LIN {X 0,Y 509.241,Z 401.693,A -85,B 0,C 180,E1 -5493.165,E2 -5493.165} C_VEL
LIN {X 0,Y 509.206,Z 398.683,A -85,B 0,C 180,E1 -5494.354,E2 -5494.354} C_VEL
LIN {X 0,Y 509.294,Z 394.619,A -85,B 0,C 180,E1 -5495.543,E2 -5495.543} C_VEL
LIN {X 0,Y 509.333,Z 388.46,A -85,B 0,C 180,E1 -5496.915,E2 -5496.915} C_VEL
LIN {X 0,Y 509.483,Z 381.524,A -85,B 0,C 180,E1 -5498.129,E2 -5498.129} C_VEL
LIN {X 0,Y 509.697,Z 373.046,A -85,B 0,C 180,E1 -5499.324,E2 -5499.324} C_VEL
LIN {X 0,Y 509.919,Z 364.313,A -85,B 0,C 180,E1 -5500.322,E2 -5500.322} C_VEL
LIN {X 0,Y 510.231,Z 353.55,A -85,B 0,C 180,E1 -5501.32,E2 -5501.32} C_VEL
LIN {X 0,Y 510.486,Z 343.069,A -85,B 0,C 180,E1 -5502.106,E2 -5502.106} C_VEL
LIN {X 0,Y 510.806,Z 331.03,A -85,B 0,C 180,E1 -5502.818,E2 -5502.818} C_VEL
LIN {X 0,Y 511.201,Z 317.442,A -85,B 0,C 180,E1 -5503.415,E2 -5503.415} C_VEL
LIN {X 0,Y 511.456,Z 304.303,A -85,B 0,C 180,E1 -5503.813,E2 -5503.813} C_VEL
LIN {X 0,Y 511.652,Z 286.942,A -85,B 0,C 180,E1 -5504.112,E2 -5504.112} C_VEL
LIN {X 0,Y 511.99,Z 204.442,A -85,B 0,C 180,E1 -5505.327,E2 -5505.327} C_VEL
LIN {X 0,Y 510.147,Z 190.872,A -85,B 0,C 180,E1 -5505.604,E2 -5505.604} C_VEL
LIN {X 0,Y 510.62,Z 169.875,A -85,B 0,C 180,E1 -5508.663,E2 -5508.663} C_VEL
LIN {X 0,Y 510.988,Z 150.072,A -85,B 0,C 180,E1 -5511.587,E2 -5511.587} C_VEL
LIN {X 0,Y 511.398,Z 134.425,A -85,B 0,C 180,E1 -5513.917,E2 -5513.917} C_VEL
LIN {X 0,Y 510.505,Z 127.875,A -85,B 0,C 180,E1 -5514.945,E2 -5514.945} C_VEL
LIN {X 0,Y 509.935,Z 124.966,A -85,B 0,C 180,E1 -5515.43,E2 -5515.43} C_VEL
LIN {X 0,Y 509.9,Z 124.975,A -85,B 0,C 180,E1 -5518.101,E2 -5518.101} C_VEL
LIN {X 0,Y 509.849,Z 124.975,A -85,B 0,C 180,E1 -5521.28,E2 -5521.28} C_VEL
LIN {X 0,Y 509.86,Z 124.978,A -85,B 0,C 180,E1 -5524.203,E2 -5524.203} C_VEL
LIN {X 0,Y 509.821,Z 124.977,A -85,B 0,C 180,E1 -5527.341,E2 -5527.341} C_VEL
LIN {X 0,Y 509.842,Z 124.978,A -85,B 0,C 180,E1 -5530.382,E2 -5530.382} C_VEL
LIN {X 0,Y 509.827,Z 124.975,A -85,B 0,C 180,E1 -5533.062,E2 -5533.062} C_VEL
LIN {X 0,Y 509.835,Z 124.98,A -85,B 0,C 180,E1 -5535.792,E2 -5535.792} C_VEL
LIN {X 0,Y 509.859,Z 124.969,A -85,B 0,C 180,E1 -5538.574,E2 -5538.574} C_VEL
LIN {X 0,Y 509.854,Z 124.977,A -85,B 0,C 180,E1 -5541.786,E2 -5541.786} C_VEL
LIN {X 0,Y 509.832,Z 124.973,A -85,B 0,C 180,E1 -5544.622,E2 -5544.622} C_VEL
LIN {X 0,Y 509.863,Z 124.977,A -85,B 0,C 180,E1 -5547.481,E2 -5547.481} C_VEL
LIN {X 0,Y 509.861,Z 124.97,A -85,B 0,C 180,E1 -5550.274,E2 -5550.274} C_VEL
LIN {X 0,Y 509.886,Z 124.971,A -85,B 0,C 180,E1 -5552.944,E2 -5552.944} C_VEL
LIN {X 0,Y 509.865,Z 124.974,A -85,B 0,C 180,E1 -5555.573,E2 -5555.573} C_VEL
LIN {X 0,Y 509.853,Z 124.978,A -85,B 0,C 180,E1 -5558.998,E2 -5558.998} C_VEL
LIN {X 0,Y 509.86,Z 124.971,A -85,B 0,C 180,E1 -5561.516,E2 -5561.516} C_VEL
LIN {X 0,Y 509.914,Z 124.969,A -85,B 0,C 180,E1 -5564.819,E2 -5564.819} C_VEL
LIN {X 0,Y 509.904,Z 124.966,A -85,B 0,C 180,E1 -5568.124,E2 -5568.124} C_VEL
LIN {X 0,Y 509.906,Z 124.969,A -85,B 0,C 180,E1 -5571.279,E2 -5571.279} C_VEL
LIN {X 0,Y 509.978,Z 124.963,A -85,B 0,C 180,E1 -5574.464,E2 -5574.464} C_VEL
LIN {X 0,Y 510.053,Z 124.949,A -85,B 0,C 180,E1 -5577.631,E2 -5577.631} C_VEL
LIN {X 0,Y 510.062,Z 124.951,A -85,B 0,C 180,E1 -5580.789,E2 -5580.789} C_VEL
LIN {X 0,Y 509.918,Z 124.967,A -85,B 0,C 180,E1 -5583.16,E2 -5583.16} C_VEL
LIN {X 0,Y 509.947,Z 124.969,A -85,B 0,C 180,E1 -5586.33,E2 -5586.33} C_VEL
LIN {X 0,Y 509.937,Z 124.998,A -85,B 0,C 180,E1 -5586.668,E2 -5586.668} C_VEL
LIN {X 0,Y 510.394,Z 130.396,A -85,B 0,C 180,E1 -5587.705,E2 -5587.705} C_VEL
LIN {X 0,Y 510.262,Z 139.77,A -85,B 0,C 180,E1 -5589.488,E2 -5589.488} C_VEL
LIN {X 0,Y 512.277,Z 149.321,A -85,B 0,C 180,E1 -5589.7,E2 -5589.7} C_VEL
LIN {X 0,Y 511.652,Z 246.787,A -85,B 0,C 180,E1 -5591.162,E2 -5591.162} C_VEL
LIN {X 0,Y 511.459,Z 260.68,A -85,B 0,C 180,E1 -5591.543,E2 -5591.543} C_VEL
LIN {X 0,Y 511.272,Z 272.633,A -85,B 0,C 180,E1 -5592.027,E2 -5592.027} C_VEL
LIN {X 0,Y 510.994,Z 283.29,A -85,B 0,C 180,E1 -5592.598,E2 -5592.598} C_VEL
LIN {X 0,Y 510.703,Z 293.998,A -85,B 0,C 180,E1 -5593.326,E2 -5593.326} C_VEL
LIN {X 0,Y 510.405,Z 304.826,A -85,B 0,C 180,E1 -5594.248,E2 -5594.248} C_VEL
LIN {X 0,Y 510.14,Z 313.67,A -85,B 0,C 180,E1 -5595.174,E2 -5595.174} C_VEL
LIN {X 0,Y 509.872,Z 321.804,A -85,B 0,C 180,E1 -5596.208,E2 -5596.208} C_VEL
LIN {X 0,Y 509.642,Z 329.686,A -85,B 0,C 180,E1 -5597.453,E2 -5597.453} C_VEL
LIN {X 0,Y 509.522,Z 335.038,A -85,B 0,C 180,E1 -5598.496,E2 -5598.496} C_VEL
LIN {X 0,Y 509.401,Z 340.193,A -85,B 0,C 180,E1 -5599.756,E2 -5599.756} C_VEL
LIN {X 0,Y 509.298,Z 344.129,A -85,B 0,C 180,E1 -5601.025,E2 -5601.025} C_VEL
LIN {X 0,Y 509.181,Z 347.04,A -85,B 0,C 180,E1 -5602.366,E2 -5602.366} C_VEL
LIN {X 0,Y 509.112,Z 348.648,A -85,B 0,C 180,E1 -5603.598,E2 -5603.598} C_VEL
LIN {X 0,Y 509.093,Z 349.21,A -85,B 0,C 180,E1 -5604.465,E2 -5604.465} C_VEL
LIN {X 0,Y 509.104,Z 349.255,A -85,B 0,C 180,E1 -5605.337,E2 -5605.337} C_VEL
LIN {X 0,Y 509.179,Z 348.845,A -85,B 0,C 180,E1 -5606.211,E2 -5606.211} C_VEL
LIN {X 0,Y 509.17,Z 347.921,A -85,B 0,C 180,E1 -5607.096,E2 -5607.096} C_VEL
LIN {X 0,Y 509.211,Z 346.477,A -85,B 0,C 180,E1 -5607.986,E2 -5607.986} C_VEL
LIN {X 0,Y 509.289,Z 343.51,A -85,B 0,C 180,E1 -5609.252,E2 -5609.252} C_VEL
LIN {X 0,Y 509.38,Z 338.713,A -85,B 0,C 180,E1 -5610.696,E2 -5610.696} C_VEL
LIN {X 0,Y 509.57,Z 332.522,A -85,B 0,C 180,E1 -5612.072,E2 -5612.072} C_VEL
LIN {X 0,Y 509.713,Z 325.689,A -85,B 0,C 180,E1 -5613.271,E2 -5613.271} C_VEL
LIN {X 0,Y 509.987,Z 317.684,A -85,B 0,C 180,E1 -5614.403,E2 -5614.403} C_VEL
LIN {X 0,Y 510.277,Z 308.043,A -85,B 0,C 180,E1 -5615.499,E2 -5615.499} C_VEL
LIN {X 0,Y 510.388,Z 303.34,A -85,B 0,C 180,E1 -5615.958,E2 -5615.958} C_VEL
LIN {X 0,Y 509.896,Z 298.789,A -85,B 0,C 180,E1 -5616.38,E2 -5616.38} C_VEL
LIN {X 0,Y 507.279,Z 291.258,A -85,B 0,C 180,E1 -5617.049,E2 -5617.049} C_VEL
LIN {X 0,Y 504.664,Z 283.306,A -85,B 0,C 180,E1 -5617.651,E2 -5617.651} C_VEL
LIN {X 0,Y 504.165,Z 278.101,A -85,B 0,C 180,E1 -5617.961,E2 -5617.961} C_VEL
LIN {X 0,Y 504.437,Z 266.65,A -85,B 0,C 180,E1 -5618.506,E2 -5618.506} C_VEL
LIN {X 0,Y 504.625,Z 253.609,A -85,B 0,C 180,E1 -5618.952,E2 -5618.952} C_VEL
LIN {X 0,Y 504.789,Z 239.971,A -85,B 0,C 180,E1 -5619.243,E2 -5619.243} C_VEL
LIN {X 0,Y 505.29,Z 149.333,A -85,B 0,C 180,E1 -5620.595,E2 -5620.595} C_VEL
LIN {X 0,Y 503.254,Z 139.407,A -85,B 0,C 180,E1 -5620.831,E2 -5620.831} C_VEL
LIN {X 0,Y 503.296,Z 128.569,A -85,B 0,C 180,E1 -5623.039,E2 -5623.039} C_VEL
LIN {X 0,Y 502.861,Z 125.85,A -85,B 0,C 180,E1 -5623.642,E2 -5623.642} C_VEL
LIN {X 0,Y 502.773,Z 125.855,A -85,B 0,C 180,E1 -5626.768,E2 -5626.768} C_VEL
LIN {X 0,Y 502.819,Z 125.848,A -85,B 0,C 180,E1 -5629.005,E2 -5629.005} C_VEL
LIN {X 0,Y 502.793,Z 125.853,A -85,B 0,C 180,E1 -5632.046,E2 -5632.046} C_VEL
LIN {X 0,Y 502.795,Z 125.852,A -85,B 0,C 180,E1 -5635.034,E2 -5635.034} C_VEL
LIN {X 0,Y 502.781,Z 125.855,A -85,B 0,C 180,E1 -5637.915,E2 -5637.915} C_VEL
LIN {X 0,Y 502.822,Z 125.847,A -85,B 0,C 180,E1 -5640.712,E2 -5640.712} C_VEL
LIN {X 0,Y 502.862,Z 125.849,A -85,B 0,C 180,E1 -5643.439,E2 -5643.439} C_VEL
LIN {X 0,Y 502.785,Z 125.852,A -85,B 0,C 180,E1 -5646.086,E2 -5646.086} C_VEL
LIN {X 0,Y 502.782,Z 125.853,A -85,B 0,C 180,E1 -5648.689,E2 -5648.689} C_VEL
LIN {X 0,Y 502.825,Z 125.854,A -85,B 0,C 180,E1 -5651.248,E2 -5651.248} C_VEL
LIN {X 0,Y 502.848,Z 125.845,A -85,B 0,C 180,E1 -5654.6,E2 -5654.6} C_VEL
LIN {X 0,Y 502.875,Z 125.84,A -85,B 0,C 180,E1 -5658.039,E2 -5658.039} C_VEL
LIN {X 0,Y 502.872,Z 125.847,A -85,B 0,C 180,E1 -5661.156,E2 -5661.156} C_VEL
LIN {X 0,Y 502.905,Z 125.837,A -85,B 0,C 180,E1 -5663.581,E2 -5663.581} C_VEL
LIN {X 0,Y 502.897,Z 125.845,A -85,B 0,C 180,E1 -5666.795,E2 -5666.795} C_VEL
LIN {X 0,Y 503.032,Z 125.824,A -85,B 0,C 180,E1 -5669.199,E2 -5669.199} C_VEL
LIN {X 0,Y 502.898,Z 125.837,A -85,B 0,C 180,E1 -5671.601,E2 -5671.601} C_VEL
LIN {X 0,Y 502.895,Z 125.84,A -85,B 0,C 180,E1 -5673.204,E2 -5673.204} C_VEL
LIN {X 0,Y 502.906,Z 125.841,A -85,B 0,C 180,E1 -5676.419,E2 -5676.419} C_VEL
LIN {X 0,Y 502.873,Z 125.846,A -85,B 0,C 180,E1 -5678.843,E2 -5678.843} C_VEL
LIN {X 0,Y 502.844,Z 125.846,A -85,B 0,C 180,E1 -5682.101,E2 -5682.101} C_VEL
LIN {X 0,Y 502.847,Z 125.843,A -85,B 0,C 180,E1 -5685.399,E2 -5685.399} C_VEL
LIN {X 0,Y 502.844,Z 125.848,A -85,B 0,C 180,E1 -5688.122,E2 -5688.122} C_VEL
LIN {X 0,Y 502.826,Z 125.852,A -85,B 0,C 180,E1 -5690.536,E2 -5690.536} C_VEL
LIN {X 0,Y 502.785,Z 125.852,A -85,B 0,C 180,E1 -5693.04,E2 -5693.04} C_VEL
LIN {X 0,Y 502.819,Z 125.848,A -85,B 0,C 180,E1 -5695.676,E2 -5695.676} C_VEL
LIN {X 0,Y 502.838,Z 125.851,A -85,B 0,C 180,E1 -5698.372,E2 -5698.372} C_VEL
LIN {X 0,Y 502.795,Z 125.851,A -85,B 0,C 180,E1 -5701.5,E2 -5701.5} C_VEL
LIN {X 0,Y 502.802,Z 125.852,A -85,B 0,C 180,E1 -5704.444,E2 -5704.444} C_VEL
LIN {X 0,Y 502.778,Z 125.852,A -85,B 0,C 180,E1 -5707.178,E2 -5707.178} C_VEL
LIN {X 0,Y 502.785,Z 125.859,A -85,B 0,C 180,E1 -5710.015,E2 -5710.015} C_VEL
LIN {X 0,Y 502.826,Z 125.85,A -85,B 0,C 180,E1 -5712.203,E2 -5712.203} C_VEL
LIN {X 0,Y 502.798,Z 125.853,A -85,B 0,C 180,E1 -5715.468,E2 -5715.468} C_VEL
LIN {X 0,Y 502.823,Z 125.847,A -85,B 0,C 180,E1 -5719.004,E2 -5719.004} C_VEL
LIN {X 0,Y 502.791,Z 125.854,A -85,B 0,C 180,E1 -5722.046,E2 -5722.046} C_VEL
LIN {X 0,Y 502.795,Z 125.851,A -85,B 0,C 180,E1 -5725.034,E2 -5725.034} C_VEL
LIN {X 0,Y 502.785,Z 125.855,A -85,B 0,C 180,E1 -5727.916,E2 -5727.916} C_VEL
LIN {X 0,Y 502.821,Z 125.847,A -85,B 0,C 180,E1 -5730.712,E2 -5730.712} C_VEL
LIN {X 0,Y 502.859,Z 125.851,A -85,B 0,C 180,E1 -5733.439,E2 -5733.439} C_VEL
LIN {X 0,Y 502.782,Z 125.852,A -85,B 0,C 180,E1 -5736.086,E2 -5736.086} C_VEL
LIN {X 0,Y 502.78,Z 125.853,A -85,B 0,C 180,E1 -5738.689,E2 -5738.689} C_VEL
LIN {X 0,Y 502.827,Z 125.854,A -85,B 0,C 180,E1 -5741.248,E2 -5741.248} C_VEL
LIN {X 0,Y 502.819,Z 125.849,A -85,B 0,C 180,E1 -5743.767,E2 -5743.767} C_VEL
LIN {X 0,Y 502.828,Z 125.846,A -85,B 0,C 180,E1 -5746.255,E2 -5746.255} C_VEL
LIN {X 0,Y 502.875,Z 125.843,A -85,B 0,C 180,E1 -5748.717,E2 -5748.717} C_VEL
LIN {X 0,Y 502.899,Z 125.837,A -85,B 0,C 180,E1 -5751.967,E2 -5751.967} C_VEL
LIN {X 0,Y 502.932,Z 125.834,A -85,B 0,C 180,E1 -5754.387,E2 -5754.387} C_VEL
LIN {X 0,Y 503.024,Z 125.822,A -85,B 0,C 180,E1 -5757.598,E2 -5757.598} C_VEL
LIN {X 0,Y 503.033,Z 125.828,A -85,B 0,C 180,E1 -5760.801,E2 -5760.801} C_VEL
LIN {X 0,Y 502.895,Z 125.84,A -85,B 0,C 180,E1 -5763.205,E2 -5763.205} C_VEL
LIN {X 0,Y 502.931,Z 125.837,A -85,B 0,C 180,E1 -5766.419,E2 -5766.419} C_VEL
LIN {X 0,Y 502.873,Z 125.846,A -85,B 0,C 180,E1 -5768.844,E2 -5768.844} C_VEL
LIN {X 0,Y 502.845,Z 125.846,A -85,B 0,C 180,E1 -5772.102,E2 -5772.102} C_VEL
LIN {X 0,Y 502.847,Z 125.843,A -85,B 0,C 180,E1 -5775.4,E2 -5775.4} C_VEL
LIN {X 0,Y 502.845,Z 125.847,A -85,B 0,C 180,E1 -5778.123,E2 -5778.123} C_VEL
LIN {X 0,Y 502.828,Z 125.853,A -85,B 0,C 180,E1 -5780.537,E2 -5780.537} C_VEL
LIN {X 0,Y 502.787,Z 125.852,A -85,B 0,C 180,E1 -5783.041,E2 -5783.041} C_VEL
LIN {X 0,Y 502.821,Z 125.848,A -85,B 0,C 180,E1 -5785.677,E2 -5785.677} C_VEL
LIN {X 0,Y 502.839,Z 125.851,A -85,B 0,C 180,E1 -5788.373,E2 -5788.373} C_VEL
LIN {X 0,Y 502.792,Z 125.851,A -85,B 0,C 180,E1 -5791.499,E2 -5791.499} C_VEL
LIN {X 0,Y 502.803,Z 125.855,A -85,B 0,C 180,E1 -5793.994,E2 -5793.994} C_VEL
LIN {X 0,Y 502.777,Z 125.852,A -85,B 0,C 180,E1 -5797.178,E2 -5797.178} C_VEL
LIN {X 0,Y 502.819,Z 125.856,A -85,B 0,C 180,E1 -5800.013,E2 -5800.013} C_VEL
LIN {X 0,Y 502.774,Z 125.853,A -85,B 0,C 180,E1 -5803.232,E2 -5803.232} C_VEL
LIN {X 0,Y 502.791,Z 125.856,A -85,B 0,C 180,E1 -5805.662,E2 -5805.662} C_VEL
LIN {X 0,Y 502.82,Z 125.847,A -85,B 0,C 180,E1 -5809.005,E2 -5809.005} C_VEL
LIN {X 0,Y 502.794,Z 125.854,A -85,B 0,C 180,E1 -5812.047,E2 -5812.047} C_VEL
LIN {X 0,Y 502.8,Z 125.85,A -85,B 0,C 180,E1 -5815.035,E2 -5815.035} C_VEL
LIN {X 0,Y 502.784,Z 125.857,A -85,B 0,C 180,E1 -5817.916,E2 -5817.916} C_VEL
LIN {X 0,Y 502.825,Z 125.847,A -85,B 0,C 180,E1 -5820.713,E2 -5820.713} C_VEL
LIN {X 0,Y 502.88,Z 125.895,A -85,B 0,C 180,E1 -5824.021,E2 -5824.021} C_VEL
LIN {X 0,Y 504.797,Z 136.242,A -85,B 0,C 180,E1 -5825.751,E2 -5825.751} C_VEL
LIN {X 0,Y 504.24,Z 155.636,A -85,B 0,C 180,E1 -5828.754,E2 -5828.754} C_VEL
LIN {X 0,Y 503.623,Z 177.725,A -85,B 0,C 180,E1 -5832.121,E2 -5832.121} C_VEL
LIN {X 0,Y 503.211,Z 191.477,A -85,B 0,C 180,E1 -5834.191,E2 -5834.191} C_VEL
LIN {X 0,Y 505.211,Z 205.925,A -85,B 0,C 180,E1 -5834.48,E2 -5834.48} C_VEL
LIN {X 0,Y 504.68,Z 301.201,A -85,B 0,C 180,E1 -5835.921,E2 -5835.921} C_VEL
LIN {X 0,Y 504.414,Z 313.294,A -85,B 0,C 180,E1 -5836.248,E2 -5836.248} C_VEL
LIN {X 0,Y 504.085,Z 326.044,A -85,B 0,C 180,E1 -5836.752,E2 -5836.752} C_VEL
LIN {X 0,Y 503.72,Z 337.99,A -85,B 0,C 180,E1 -5837.394,E2 -5837.394} C_VEL
LIN {X 0,Y 503.312,Z 349.792,A -85,B 0,C 180,E1 -5838.217,E2 -5838.217} C_VEL
LIN {X 0,Y 503.048,Z 360.245,A -85,B 0,C 180,E1 -5839.129,E2 -5839.129} C_VEL
LIN {X 0,Y 502.717,Z 369.632,A -85,B 0,C 180,E1 -5840.14,E2 -5840.14} C_VEL
LIN {X 0,Y 502.474,Z 378.731,A -85,B 0,C 180,E1 -5841.353,E2 -5841.353} C_VEL
LIN {X 0,Y 502.313,Z 386.062,A -85,B 0,C 180,E1 -5842.564,E2 -5842.564} C_VEL
LIN {X 0,Y 502.216,Z 391.012,A -85,B 0,C 180,E1 -5843.572,E2 -5843.572} C_VEL
LIN {X 0,Y 502.176,Z 395.818,A -85,B 0,C 180,E1 -5844.781,E2 -5844.781} C_VEL
LIN {X 0,Y 502.165,Z 399.489,A -85,B 0,C 180,E1 -5845.988,E2 -5845.988} C_VEL
LIN {X 0,Y 502.158,Z 401.381,A -85,B 0,C 180,E1 -5846.791,E2 -5846.791} C_VEL
LIN {X 0,Y 502.128,Z 402.799,A -85,B 0,C 180,E1 -5847.594,E2 -5847.594} C_VEL
LIN {X 0,Y 502.009,Z 404.407,A -85,B 0,C 180,E1 -5849.198,E2 -5849.198} C_VEL
LIN {X 0,Y 502.01,Z 404.617,A -85,B 0,C 180,E1 -5850,E2 -5850} C_VEL
LIN {X 0,Y 502.01,Z 404.386,A -85,B 0,C 180,E1 -5850.802,E2 -5850.802} C_VEL
LIN {X 0,Y 502.128,Z 402.729,A -85,B 0,C 180,E1 -5852.407,E2 -5852.407} C_VEL
LIN {X 0,Y 502.158,Z 401.289,A -85,B 0,C 180,E1 -5853.21,E2 -5853.21} C_VEL
LIN {X 0,Y 502.104,Z 398.268,A -85,B 0,C 180,E1 -5854.416,E2 -5854.416} C_VEL
LIN {X 0,Y 502.202,Z 394.19,A -85,B 0,C 180,E1 -5855.622,E2 -5855.622} C_VEL
LIN {X 0,Y 502.274,Z 388.01,A -85,B 0,C 180,E1 -5857.013,E2 -5857.013} C_VEL
LIN {X 0,Y 502.42,Z 381.054,A -85,B 0,C 180,E1 -5858.244,E2 -5858.244} C_VEL
LIN {X 0,Y 502.647,Z 372.554,A -85,B 0,C 180,E1 -5859.456,E2 -5859.456} C_VEL
LIN {X 0,Y 502.913,Z 363.795,A -85,B 0,C 180,E1 -5860.467,E2 -5860.467} C_VEL
LIN {X 0,Y 503.172,Z 353.001,A -85,B 0,C 180,E1 -5861.481,E2 -5861.481} C_VEL
LIN {X 0,Y 503.515,Z 342.196,A -85,B 0,C 180,E1 -5862.297,E2 -5862.297} C_VEL
LIN {X 0,Y 503.868,Z 330.394,A -85,B 0,C 180,E1 -5862.998,E2 -5862.998} C_VEL
LIN {X 0,Y 504.227,Z 318.046,A -85,B 0,C 180,E1 -5863.553,E2 -5863.553} C_VEL
LIN {X 0,Y 504.528,Z 304.531,A -85,B 0,C 180,E1 -5863.981,E2 -5863.981} C_VEL
LIN {X 0,Y 504.729,Z 289.383,A -85,B 0,C 180,E1 -5864.258,E2 -5864.258} C_VEL
LIN {X 0,Y 505.125,Z 205.087,A -85,B 0,C 180,E1 -5865.527,E2 -5865.527} C_VEL
LIN {X 0,Y 503.155,Z 190.339,A -85,B 0,C 180,E1 -5865.84,E2 -5865.84} C_VEL
LIN {X 0,Y 503.658,Z 169.471,A -85,B 0,C 180,E1 -5868.931,E2 -5868.931} C_VEL
LIN {X 0,Y 504.022,Z 151.067,A -85,B 0,C 180,E1 -5871.686,E2 -5871.686} C_VEL
LIN {X 0,Y 504.469,Z 135.425,A -85,B 0,C 180,E1 -5874.048,E2 -5874.048} C_VEL
LIN {X 0,Y 503.053,Z 126.745,A -85,B 0,C 180,E1 -5875.453,E2 -5875.453} C_VEL
LIN {X 0,Y 502.9,Z 125.843,A -85,B 0,C 180,E1 -5875.62,E2 -5875.62} C_VEL
LIN {X 0,Y 502.844,Z 125.856,A -85,B 0,C 180,E1 -5878.373,E2 -5878.373} C_VEL
LIN {X 0,Y 502.797,Z 125.854,A -85,B 0,C 180,E1 -5881.499,E2 -5881.499} C_VEL
LIN {X 0,Y 502.808,Z 125.856,A -85,B 0,C 180,E1 -5883.994,E2 -5883.994} C_VEL
LIN {X 0,Y 502.781,Z 125.853,A -85,B 0,C 180,E1 -5887.178,E2 -5887.178} C_VEL
LIN {X 0,Y 502.791,Z 125.858,A -85,B 0,C 180,E1 -5890.015,E2 -5890.015} C_VEL
LIN {X 0,Y 502.807,Z 125.855,A -85,B 0,C 180,E1 -5892.199,E2 -5892.199} C_VEL
LIN {X 0,Y 502.805,Z 125.853,A -85,B 0,C 180,E1 -5895.468,E2 -5895.468} C_VEL
LIN {X 0,Y 502.823,Z 125.845,A -85,B 0,C 180,E1 -5898.934,E2 -5898.934} C_VEL
LIN {X 0,Y 502.796,Z 125.852,A -85,B 0,C 180,E1 -5902.046,E2 -5902.046} C_VEL
LIN {X 0,Y 502.798,Z 125.851,A -85,B 0,C 180,E1 -5905.034,E2 -5905.034} C_VEL
LIN {X 0,Y 502.785,Z 125.852,A -85,B 0,C 180,E1 -5907.915,E2 -5907.915} C_VEL
LIN {X 0,Y 502.826,Z 125.848,A -85,B 0,C 180,E1 -5910.712,E2 -5910.712} C_VEL
LIN {X 0,Y 502.866,Z 125.846,A -85,B 0,C 180,E1 -5913.439,E2 -5913.439} C_VEL
LIN {X 0,Y 502.787,Z 125.852,A -85,B 0,C 180,E1 -5916.086,E2 -5916.086} C_VEL
LIN {X 0,Y 502.786,Z 125.854,A -85,B 0,C 180,E1 -5918.689,E2 -5918.689} C_VEL
LIN {X 0,Y 502.825,Z 125.851,A -85,B 0,C 180,E1 -5921.248,E2 -5921.248} C_VEL
LIN {X 0,Y 502.852,Z 125.847,A -85,B 0,C 180,E1 -5924.6,E2 -5924.6} C_VEL
LIN {X 0,Y 502.88,Z 125.841,A -85,B 0,C 180,E1 -5928.039,E2 -5928.039} C_VEL
LIN {X 0,Y 502.866,Z 125.847,A -85,B 0,C 180,E1 -5931.156,E2 -5931.156} C_VEL
LIN {X 0,Y 502.931,Z 125.841,A -85,B 0,C 180,E1 -5934.386,E2 -5934.386} C_VEL
LIN {X 0,Y 503.022,Z 125.825,A -85,B 0,C 180,E1 -5937.597,E2 -5937.597} C_VEL
LIN {X 0,Y 503.012,Z 125.83,A -85,B 0,C 180,E1 -5940.8,E2 -5940.8} C_VEL
LIN {X 0,Y 503.019,Z 125.831,A -85,B 0,C 180,E1 -5942.402,E2 -5942.402} C_VEL
LIN {X 0,Y 502.929,Z 125.838,A -85,B 0,C 180,E1 -5945.613,E2 -5945.613} C_VEL
LIN {X 0,Y 502.915,Z 125.921,A -85,B 0,C 180,E1 -5946.521,E2 -5946.521} C_VEL
LIN {X 0,Y 503.441,Z 131.586,A -85,B 0,C 180,E1 -5947.625,E2 -5947.625} C_VEL
LIN {X 0,Y 503.331,Z 140.147,A -85,B 0,C 180,E1 -5949.255,E2 -5949.255} C_VEL
LIN {X 0,Y 505.513,Z 151.243,A -85,B 0,C 180,E1 -5949.51,E2 -5949.51} C_VEL
LIN {X 0,Y 504.767,Z 247.615,A -85,B 0,C 180,E1 -5950.986,E2 -5950.986} C_VEL
LIN {X 0,Y 504.562,Z 261.351,A -85,B 0,C 180,E1 -5951.372,E2 -5951.372} C_VEL
LIN {X 0,Y 504.351,Z 274.181,A -85,B 0,C 180,E1 -5951.912,E2 -5951.912} C_VEL
LIN {X 0,Y 504.023,Z 285.668,A -85,B 0,C 180,E1 -5952.56,E2 -5952.56} C_VEL
LIN {X 0,Y 503.686,Z 297.456,A -85,B 0,C 180,E1 -5953.413,E2 -5953.413} C_VEL
LIN {X 0,Y 503.339,Z 307.699,A -85,B 0,C 180,E1 -5954.349,E2 -5954.349} C_VEL
LIN {X 0,Y 503.05,Z 317.185,A -85,B 0,C 180,E1 -5955.423,E2 -5955.423} C_VEL
LIN {X 0,Y 502.737,Z 325.95,A -85,B 0,C 180,E1 -5956.653,E2 -5956.653} C_VEL
LIN {X 0,Y 502.513,Z 333.505,A -85,B 0,C 180,E1 -5958.005,E2 -5958.005} C_VEL
LIN {X 0,Y 502.408,Z 338.747,A -85,B 0,C 180,E1 -5959.192,E2 -5959.192} C_VEL
LIN {X 0,Y 502.265,Z 343.157,A -85,B 0,C 180,E1 -5960.476,E2 -5960.476} C_VEL
LIN {X 0,Y 502.193,Z 345.44,A -85,B 0,C 180,E1 -5961.337,E2 -5961.337} C_VEL
LIN {X 0,Y 502.086,Z 347.736,A -85,B 0,C 180,E1 -5962.505,E2 -5962.505} C_VEL
LIN {X 0,Y 502.019,Z 349.328,A -85,B 0,C 180,E1 -5963.952,E2 -5963.952} C_VEL
LIN {X 0,Y 502.006,Z 349.667,A -85,B 0,C 180,E1 -5964.834,E2 -5964.834} C_VEL
LIN {X 0,Y 502.103,Z 349.111,A -85,B 0,C 180,E1 -5966.386,E2 -5966.386} C_VEL
LIN {X 0,Y 502.098,Z 347.754,A -85,B 0,C 180,E1 -5967.51,E2 -5967.51} C_VEL
LIN {X 0,Y 502.185,Z 345.046,A -85,B 0,C 180,E1 -5968.87,E2 -5968.87} C_VEL
LIN {X 0,Y 502.261,Z 340.98,A -85,B 0,C 180,E1 -5970.247,E2 -5970.247} C_VEL
LIN {X 0,Y 502.468,Z 335.01,A -85,B 0,C 180,E1 -5971.728,E2 -5971.728} C_VEL
LIN {X 0,Y 502.652,Z 328.088,A -85,B 0,C 180,E1 -5973.044,E2 -5973.044} C_VEL
LIN {X 0,Y 502.91,Z 320.228,A -85,B 0,C 180,E1 -5974.231,E2 -5974.231} C_VEL
LIN {X 0,Y 503.169,Z 311.517,A -85,B 0,C 180,E1 -5975.303,E2 -5975.303} C_VEL
LIN {X 0,Y 503.516,Z 301.138,A -85,B 0,C 180,E1 -5976.335,E2 -5976.335} C_VEL
LIN {X 0,Y 503.866,Z 290.01,A -85,B 0,C 180,E1 -5977.216,E2 -5977.216} C_VEL
LIN {X 0,Y 504.165,Z 278.101,A -85,B 0,C 180,E1 -5977.961,E2 -5977.961} C_VEL
LIN {X 0,Y 503.734,Z 272.774,A -85,B 0,C 180,E1 -5978.25,E2 -5978.25} C_VEL
LIN {X 0,Y 501.179,Z 264.065,A -85,B 0,C 180,E1 -5978.7,E2 -5978.7} C_VEL
LIN {X 0,Y 498.517,Z 255.135,A -85,B 0,C 180,E1 -5979.083,E2 -5979.083} C_VEL
LIN {X 0,Y 497.825,Z 249.464,A -85,B 0,C 180,E1 -5979.252,E2 -5979.252} C_VEL
LIN {X 0,Y 497.981,Z 229.704,A -85,B 0,C 180,E1 -5979.59,E2 -5979.59} C_VEL
LIN {X 0,Y 498.535,Z 150.806,A -85,B 0,C 180,E1 -5980.789,E2 -5980.789} C_VEL
LIN {X 0,Y 496.304,Z 139.721,A -85,B 0,C 180,E1 -5981.05,E2 -5981.05} C_VEL
LIN {X 0,Y 496.293,Z 129.397,A -85,B 0,C 180,E1 -5983.173,E2 -5983.173} C_VEL
LIN {X 0,Y 495.817,Z 126.728,A -85,B 0,C 180,E1 -5983.762,E2 -5983.762} C_VEL
LIN {X 0,Y 495.726,Z 126.734,A -85,B 0,C 180,E1 -5987.117,E2 -5987.117} C_VEL
LIN {X 0,Y 495.758,Z 126.731,A -85,B 0,C 180,E1 -5989.953,E2 -5989.953} C_VEL
LIN {X 0,Y 495.727,Z 126.73,A -85,B 0,C 180,E1 -5992.553,E2 -5992.553} C_VEL
LIN {X 0,Y 495.77,Z 126.732,A -85,B 0,C 180,E1 -5995.456,E2 -5995.456} C_VEL
LIN {X 0,Y 495.753,Z 126.727,A -85,B 0,C 180,E1 -5998.363,E2 -5998.363} C_VEL
LIN {X 0,Y 495.786,Z 126.73,A -85,B 0,C 180,E1 -6001.507,E2 -6001.507} C_VEL
LIN {X 0,Y 495.79,Z 126.724,A -85,B 0,C 180,E1 -6003.932,E2 -6003.932} C_VEL
LIN {X 0,Y 495.759,Z 126.732,A -85,B 0,C 180,E1 -6007.139,E2 -6007.139} C_VEL
LIN {X 0,Y 495.77,Z 126.725,A -85,B 0,C 180,E1 -6010.109,E2 -6010.109} C_VEL
LIN {X 0,Y 495.764,Z 126.728,A -85,B 0,C 180,E1 -6012.68,E2 -6012.68} C_VEL
LIN {X 0,Y 495.789,Z 126.73,A -85,B 0,C 180,E1 -6015.217,E2 -6015.217} C_VEL
LIN {X 0,Y 495.851,Z 126.717,A -85,B 0,C 180,E1 -6018.555,E2 -6018.555} C_VEL
LIN {X 0,Y 495.872,Z 126.712,A -85,B 0,C 180,E1 -6021.852,E2 -6021.852} C_VEL
LIN {X 0,Y 495.888,Z 126.711,A -85,B 0,C 180,E1 -6024.306,E2 -6024.306} C_VEL
LIN {X 0,Y 495.993,Z 126.698,A -85,B 0,C 180,E1 -6027.563,E2 -6027.563} C_VEL
LIN {X 0,Y 495.998,Z 126.697,A -85,B 0,C 180,E1 -6030,E2 -6030} C_VEL
LIN {X 0,Y 495.993,Z 126.701,A -85,B 0,C 180,E1 -6032.436,E2 -6032.436} C_VEL
LIN {X 0,Y 495.889,Z 126.71,A -85,B 0,C 180,E1 -6035.693,E2 -6035.693} C_VEL
LIN {X 0,Y 495.872,Z 126.715,A -85,B 0,C 180,E1 -6038.148,E2 -6038.148} C_VEL
LIN {X 0,Y 495.85,Z 126.715,A -85,B 0,C 180,E1 -6041.445,E2 -6041.445} C_VEL
LIN {X 0,Y 495.793,Z 126.727,A -85,B 0,C 180,E1 -6044.782,E2 -6044.782} C_VEL
LIN {X 0,Y 495.784,Z 126.723,A -85,B 0,C 180,E1 -6047.318,E2 -6047.318} C_VEL
LIN {X 0,Y 495.775,Z 126.726,A -85,B 0,C 180,E1 -6049.89,E2 -6049.89} C_VEL
LIN {X 0,Y 495.756,Z 126.728,A -85,B 0,C 180,E1 -6052.86,E2 -6052.86} C_VEL
LIN {X 0,Y 495.778,Z 126.73,A -85,B 0,C 180,E1 -6056.068,E2 -6056.068} C_VEL
LIN {X 0,Y 495.775,Z 126.725,A -85,B 0,C 180,E1 -6058.814,E2 -6058.814} C_VEL
LIN {X 0,Y 495.757,Z 126.73,A -85,B 0,C 180,E1 -6061.726,E2 -6061.726} C_VEL
LIN {X 0,Y 495.772,Z 126.726,A -85,B 0,C 180,E1 -6064.695,E2 -6064.695} C_VEL
LIN {X 0,Y 495.728,Z 126.733,A -85,B 0,C 180,E1 -6067.561,E2 -6067.561} C_VEL
LIN {X 0,Y 495.764,Z 126.726,A -85,B 0,C 180,E1 -6070.7,E2 -6070.7} C_VEL
LIN {X 0,Y 495.731,Z 126.736,A -85,B 0,C 180,E1 -6073.695,E2 -6073.695} C_VEL
LIN {X 0,Y 495.725,Z 126.733,A -85,B 0,C 180,E1 -6076.305,E2 -6076.305} C_VEL
LIN {X 0,Y 495.777,Z 126.727,A -85,B 0,C 180,E1 -6079.302,E2 -6079.302} C_VEL
LIN {X 0,Y 495.726,Z 126.731,A -85,B 0,C 180,E1 -6082.438,E2 -6082.438} C_VEL
LIN {X 0,Y 495.774,Z 126.731,A -85,B 0,C 180,E1 -6085.457,E2 -6085.457} C_VEL
LIN {X 0,Y 495.756,Z 126.727,A -85,B 0,C 180,E1 -6088.364,E2 -6088.364} C_VEL
LIN {X 0,Y 495.785,Z 126.732,A -85,B 0,C 180,E1 -6091.507,E2 -6091.507} C_VEL
LIN {X 0,Y 495.787,Z 126.725,A -85,B 0,C 180,E1 -6093.932,E2 -6093.932} C_VEL
LIN {X 0,Y 495.757,Z 126.732,A -85,B 0,C 180,E1 -6097.139,E2 -6097.139} C_VEL
LIN {X 0,Y 495.775,Z 126.725,A -85,B 0,C 180,E1 -6100.11,E2 -6100.11} C_VEL
LIN {X 0,Y 495.784,Z 126.725,A -85,B 0,C 180,E1 -6102.682,E2 -6102.682} C_VEL
LIN {X 0,Y 495.787,Z 126.731,A -85,B 0,C 180,E1 -6105.217,E2 -6105.217} C_VEL
LIN {X 0,Y 495.849,Z 126.717,A -85,B 0,C 180,E1 -6108.555,E2 -6108.555} C_VEL
LIN {X 0,Y 495.871,Z 126.713,A -85,B 0,C 180,E1 -6111.852,E2 -6111.852} C_VEL
LIN {X 0,Y 495.888,Z 126.711,A -85,B 0,C 180,E1 -6114.307,E2 -6114.307} C_VEL
LIN {X 0,Y 495.992,Z 126.698,A -85,B 0,C 180,E1 -6117.564,E2 -6117.564} C_VEL
LIN {X 0,Y 495.997,Z 126.697,A -85,B 0,C 180,E1 -6120,E2 -6120} C_VEL
LIN {X 0,Y 495.993,Z 126.701,A -85,B 0,C 180,E1 -6122.437,E2 -6122.437} C_VEL
LIN {X 0,Y 495.897,Z 126.709,A -85,B 0,C 180,E1 -6125.694,E2 -6125.694} C_VEL
LIN {X 0,Y 495.872,Z 126.714,A -85,B 0,C 180,E1 -6128.148,E2 -6128.148} C_VEL
LIN {X 0,Y 495.85,Z 126.715,A -85,B 0,C 180,E1 -6131.446,E2 -6131.446} C_VEL
LIN {X 0,Y 495.793,Z 126.727,A -85,B 0,C 180,E1 -6134.783,E2 -6134.783} C_VEL
LIN {X 0,Y 495.797,Z 126.726,A -85,B 0,C 180,E1 -6138.171,E2 -6138.171} C_VEL
LIN {X 0,Y 495.773,Z 126.729,A -85,B 0,C 180,E1 -6140.757,E2 -6140.757} C_VEL
LIN {X 0,Y 495.742,Z 126.728,A -85,B 0,C 180,E1 -6143.388,E2 -6143.388} C_VEL
LIN {X 0,Y 495.822,Z 126.721,A -85,B 0,C 180,E1 -6146.75,E2 -6146.75} C_VEL
LIN {X 0,Y 495.765,Z 126.728,A -85,B 0,C 180,E1 -6149.747,E2 -6149.747} C_VEL
LIN {X 0,Y 495.767,Z 126.728,A -85,B 0,C 180,E1 -6152.595,E2 -6152.595} C_VEL
LIN {X 0,Y 495.747,Z 126.729,A -85,B 0,C 180,E1 -6155.538,E2 -6155.538} C_VEL
LIN {X 0,Y 495.768,Z 126.726,A -85,B 0,C 180,E1 -6158.769,E2 -6158.769} C_VEL
LIN {X 0,Y 495.759,Z 126.732,A -85,B 0,C 180,E1 -6161.781,E2 -6161.781} C_VEL
LIN {X 0,Y 495.75,Z 126.728,A -85,B 0,C 180,E1 -6165.14,E2 -6165.14} C_VEL
LIN {X 0,Y 495.759,Z 126.73,A -85,B 0,C 180,E1 -6168.22,E2 -6168.22} C_VEL
LIN {X 0,Y 495.752,Z 126.731,A -85,B 0,C 180,E1 -6171.409,E2 -6171.409} C_VEL
LIN {X 0,Y 495.749,Z 126.728,A -85,B 0,C 180,E1 -6174.463,E2 -6174.463} C_VEL
LIN {X 0,Y 495.768,Z 126.73,A -85,B 0,C 180,E1 -6177.406,E2 -6177.406} C_VEL
LIN {X 0,Y 495.768,Z 126.727,A -85,B 0,C 180,E1 -6180.254,E2 -6180.254} C_VEL
LIN {X 0,Y 495.844,Z 126.724,A -85,B 0,C 180,E1 -6183.527,E2 -6183.527} C_VEL
LIN {X 0,Y 495.851,Z 126.792,A -85,B 0,C 180,E1 -6183.834,E2 -6183.834} C_VEL
LIN {X 0,Y 497.836,Z 137.263,A -85,B 0,C 180,E1 -6185.612,E2 -6185.612} C_VEL
LIN {X 0,Y 497.357,Z 153.876,A -85,B 0,C 180,E1 -6188.227,E2 -6188.227} C_VEL
LIN {X 0,Y 496.69,Z 175.427,A -85,B 0,C 180,E1 -6191.563,E2 -6191.563} C_VEL
LIN {X 0,Y 496.213,Z 191.135,A -85,B 0,C 180,E1 -6193.966,E2 -6193.966} C_VEL
LIN {X 0,Y 498.393,Z 207.837,A -85,B 0,C 180,E1 -6194.302,E2 -6194.302} C_VEL
LIN {X 0,Y 497.798,Z 300.306,A -85,B 0,C 180,E1 -6195.722,E2 -6195.722} C_VEL
LIN {X 0,Y 497.499,Z 312.558,A -85,B 0,C 180,E1 -6196.053,E2 -6196.053} C_VEL
LIN {X 0,Y 497.148,Z 325.394,A -85,B 0,C 180,E1 -6196.564,E2 -6196.564} C_VEL
LIN {X 0,Y 496.77,Z 336.313,A -85,B 0,C 180,E1 -6197.146,E2 -6197.146} C_VEL
LIN {X 0,Y 496.388,Z 347.963,A -85,B 0,C 180,E1 -6197.946,E2 -6197.946} C_VEL
LIN {X 0,Y 496.059,Z 358.669,A -85,B 0,C 180,E1 -6198.87,E2 -6198.87} C_VEL
LIN {X 0,Y 495.747,Z 367.419,A -85,B 0,C 180,E1 -6199.793,E2 -6199.793} C_VEL
LIN {X 0,Y 495.508,Z 375.483,A -85,B 0,C 180,E1 -6200.819,E2 -6200.819} C_VEL
LIN {X 0,Y 495.308,Z 383.376,A -85,B 0,C 180,E1 -6202.048,E2 -6202.048} C_VEL
LIN {X 0,Y 495.128,Z 390.601,A -85,B 0,C 180,E1 -6203.48,E2 -6203.48} C_VEL
LIN {X 0,Y 495.106,Z 395.419,A -85,B 0,C 180,E1 -6204.706,E2 -6204.706} C_VEL
LIN {X 0,Y 495.056,Z 399.096,A -85,B 0,C 180,E1 -6205.93,E2 -6205.93} C_VEL
LIN {X 0,Y 495.077,Z 400.993,A -85,B 0,C 180,E1 -6206.745,E2 -6206.745} C_VEL
LIN {X 0,Y 495.062,Z 402.413,A -85,B 0,C 180,E1 -6207.559,E2 -6207.559} C_VEL
LIN {X 0,Y 494.928,Z 404.021,A -85,B 0,C 180,E1 -6209.187,E2 -6209.187} C_VEL
LIN {X 0,Y 494.926,Z 404.23,A -85,B 0,C 180,E1 -6210,E2 -6210} C_VEL
LIN {X 0,Y 494.929,Z 403.995,A -85,B 0,C 180,E1 -6210.814,E2 -6210.814} C_VEL
LIN {X 0,Y 495.062,Z 402.333,A -85,B 0,C 180,E1 -6212.441,E2 -6212.441} C_VEL
LIN {X 0,Y 495.077,Z 400.886,A -85,B 0,C 180,E1 -6213.255,E2 -6213.255} C_VEL
LIN {X 0,Y 495.01,Z 397.854,A -85,B 0,C 180,E1 -6214.479,E2 -6214.479} C_VEL
LIN {X 0,Y 495.11,Z 393.764,A -85,B 0,C 180,E1 -6215.703,E2 -6215.703} C_VEL
LIN {X 0,Y 495.195,Z 387.464,A -85,B 0,C 180,E1 -6217.134,E2 -6217.134} C_VEL
LIN {X 0,Y 495.345,Z 380.594,A -85,B 0,C 180,E1 -6218.362,E2 -6218.362} C_VEL
LIN {X 0,Y 495.572,Z 372.067,A -85,B 0,C 180,E1 -6219.592,E2 -6219.592} C_VEL
LIN {X 0,Y 495.883,Z 363.282,A -85,B 0,C 180,E1 -6220.617,E2 -6220.617} C_VEL
LIN {X 0,Y 496.185,Z 352.469,A -85,B 0,C 180,E1 -6221.645,E2 -6221.645} C_VEL
LIN {X 0,Y 496.551,Z 340.757,A -85,B 0,C 180,E1 -6222.533,E2 -6222.533} C_VEL
LIN {X 0,Y 496.987,Z 328.808,A -85,B 0,C 180,E1 -6223.233,E2 -6223.233} C_VEL
LIN {X 0,Y 497.355,Z 316.129,A -85,B 0,C 180,E1 -6223.796,E2 -6223.796} C_VEL
LIN {X 0,Y 497.62,Z 303.836,A -85,B 0,C 180,E1 -6224.179,E2 -6224.179} C_VEL
LIN {X 0,Y 497.829,Z 288.573,A -85,B 0,C 180,E1 -6224.46,E2 -6224.46} C_VEL
LIN {X 0,Y 498.321,Z 206.036,A -85,B 0,C 180,E1 -6225.728,E2 -6225.728} C_VEL
LIN {X 0,Y 496.162,Z 189.897,A -85,B 0,C 180,E1 -6226.077,E2 -6226.077} C_VEL
LIN {X 0,Y 496.662,Z 169.05,A -85,B 0,C 180,E1 -6229.208,E2 -6229.208} C_VEL
LIN {X 0,Y 497.065,Z 152.078,A -85,B 0,C 180,E1 -6231.787,E2 -6231.787} C_VEL
LIN {X 0,Y 497.541,Z 136.487,A -85,B 0,C 180,E1 -6234.182,E2 -6234.182} C_VEL
LIN {X 0,Y 495.851,Z 126.722,A -85,B 0,C 180,E1 -6235.811,E2 -6235.811} C_VEL
LIN {X 0,Y 495.776,Z 126.734,A -85,B 0,C 180,E1 -6238.815,E2 -6238.815} C_VEL
LIN {X 0,Y 495.759,Z 126.733,A -85,B 0,C 180,E1 -6241.725,E2 -6241.725} C_VEL
LIN {X 0,Y 495.772,Z 126.729,A -85,B 0,C 180,E1 -6244.694,E2 -6244.694} C_VEL
LIN {X 0,Y 495.733,Z 126.733,A -85,B 0,C 180,E1 -6247.562,E2 -6247.562} C_VEL
LIN {X 0,Y 495.77,Z 126.728,A -85,B 0,C 180,E1 -6250.7,E2 -6250.7} C_VEL
LIN {X 0,Y 495.738,Z 126.735,A -85,B 0,C 180,E1 -6254.001,E2 -6254.001} C_VEL
LIN {X 0,Y 495.73,Z 126.731,A -85,B 0,C 180,E1 -6257.117,E2 -6257.117} C_VEL
LIN {X 0,Y 495.762,Z 126.73,A -85,B 0,C 180,E1 -6259.953,E2 -6259.953} C_VEL
LIN {X 0,Y 495.731,Z 126.729,A -85,B 0,C 180,E1 -6262.553,E2 -6262.553} C_VEL
LIN {X 0,Y 495.774,Z 126.73,A -85,B 0,C 180,E1 -6265.456,E2 -6265.456} C_VEL
LIN {X 0,Y 495.757,Z 126.725,A -85,B 0,C 180,E1 -6268.364,E2 -6268.364} C_VEL
LIN {X 0,Y 495.79,Z 126.728,A -85,B 0,C 180,E1 -6271.507,E2 -6271.507} C_VEL
LIN {X 0,Y 495.793,Z 126.722,A -85,B 0,C 180,E1 -6273.932,E2 -6273.932} C_VEL
LIN {X 0,Y 495.763,Z 126.731,A -85,B 0,C 180,E1 -6277.139,E2 -6277.139} C_VEL
LIN {X 0,Y 495.771,Z 126.725,A -85,B 0,C 180,E1 -6280.109,E2 -6280.109} C_VEL
LIN {X 0,Y 495.759,Z 126.729,A -85,B 0,C 180,E1 -6282.68,E2 -6282.68} C_VEL
LIN {X 0,Y 495.79,Z 126.729,A -85,B 0,C 180,E1 -6285.217,E2 -6285.217} C_VEL
LIN {X 0,Y 495.854,Z 126.721,A -85,B 0,C 180,E1 -6288.555,E2 -6288.555} C_VEL
LIN {X 0,Y 495.839,Z 126.719,A -85,B 0,C 180,E1 -6291.851,E2 -6291.851} C_VEL
LIN {X 0,Y 495.886,Z 126.717,A -85,B 0,C 180,E1 -6294.306,E2 -6294.306} C_VEL
LIN {X 0,Y 495.989,Z 126.701,A -85,B 0,C 180,E1 -6297.563,E2 -6297.563} C_VEL
LIN {X 0,Y 495.963,Z 126.708,A -85,B 0,C 180,E1 -6300.812,E2 -6300.812} C_VEL
LIN {X 0,Y 495.987,Z 126.707,A -85,B 0,C 180,E1 -6302.436,E2 -6302.436} C_VEL
LIN {X 0,Y 495.88,Z 126.833,A -85,B 0,C 180,E1 -6306.357,E2 -6306.357} C_VEL
LIN {X 0,Y 496.47,Z 131.703,A -85,B 0,C 180,E1 -6307.319,E2 -6307.319} C_VEL
LIN {X 0,Y 496.422,Z 140.794,A -85,B 0,C 180,E1 -6309.029,E2 -6309.029} C_VEL
LIN {X 0,Y 498.73,Z 152.384,A -85,B 0,C 180,E1 -6309.296,E2 -6309.296} C_VEL
LIN {X 0,Y 497.896,Z 247.408,A -85,B 0,C 180,E1 -6310.779,E2 -6310.779} C_VEL
LIN {X 0,Y 497.678,Z 261.317,A -85,B 0,C 180,E1 -6311.17,E2 -6311.17} C_VEL
LIN {X 0,Y 497.439,Z 274.311,A -85,B 0,C 180,E1 -6311.718,E2 -6311.718} C_VEL
LIN {X 0,Y 497.1,Z 286.518,A -85,B 0,C 180,E1 -6312.419,E2 -6312.419} C_VEL
LIN {X 0,Y 496.751,Z 297.031,A -85,B 0,C 180,E1 -6313.187,E2 -6313.187} C_VEL
LIN {X 0,Y 496.403,Z 307.46,A -85,B 0,C 180,E1 -6314.136,E2 -6314.136} C_VEL
LIN {X 0,Y 496.098,Z 316.458,A -85,B 0,C 180,E1 -6315.15,E2 -6315.15} C_VEL
LIN {X 0,Y 495.787,Z 324.52,A -85,B 0,C 180,E1 -6316.258,E2 -6316.258} C_VEL
LIN {X 0,Y 495.537,Z 331.979,A -85,B 0,C 180,E1 -6317.524,E2 -6317.524} C_VEL
LIN {X 0,Y 495.4,Z 337.128,A -85,B 0,C 180,E1 -6318.614,E2 -6318.614} C_VEL
LIN {X 0,Y 495.256,Z 342.02,A -85,B 0,C 180,E1 -6319.912,E2 -6319.912} C_VEL
LIN {X 0,Y 495.139,Z 345.689,A -85,B 0,C 180,E1 -6321.219,E2 -6321.219} C_VEL
LIN {X 0,Y 495.014,Z 348.384,A -85,B 0,C 180,E1 -6322.654,E2 -6322.654} C_VEL
LIN {X 0,Y 494.963,Z 349.303,A -85,B 0,C 180,E1 -6323.426,E2 -6323.426} C_VEL
LIN {X 0,Y 494.92,Z 350.027,A -85,B 0,C 180,E1 -6324.657,E2 -6324.657} C_VEL
LIN {X 0,Y 494.995,Z 349.695,A -85,B 0,C 180,E1 -6326.113,E2 -6326.113} C_VEL
LIN {X 0,Y 495.011,Z 348.862,A -85,B 0,C 180,E1 -6327.021,E2 -6327.021} C_VEL
LIN {X 0,Y 495.058,Z 346.719,A -85,B 0,C 180,E1 -6328.336,E2 -6328.336} C_VEL
LIN {X 0,Y 495.206,Z 343.047,A -85,B 0,C 180,E1 -6329.783,E2 -6329.783} C_VEL
LIN {X 0,Y 495.281,Z 338.09,A -85,B 0,C 180,E1 -6331.188,E2 -6331.188} C_VEL
LIN {X 0,Y 495.522,Z 332.683,A -85,B 0,C 180,E1 -6332.371,E2 -6332.371} C_VEL
LIN {X 0,Y 495.688,Z 325.912,A -85,B 0,C 180,E1 -6333.569,E2 -6333.569} C_VEL
LIN {X 0,Y 496.051,Z 316.806,A -85,B 0,C 180,E1 -6334.849,E2 -6334.849} C_VEL
LIN {X 0,Y 496.368,Z 306.995,A -85,B 0,C 180,E1 -6335.959,E2 -6335.959} C_VEL
LIN {X 0,Y 496.677,Z 297.354,A -85,B 0,C 180,E1 -6336.841,E2 -6336.841} C_VEL
LIN {X 0,Y 497.079,Z 285.362,A -85,B 0,C 180,E1 -6337.715,E2 -6337.715} C_VEL
LIN {X 0,Y 497.395,Z 273.603,A -85,B 0,C 180,E1 -6338.383,E2 -6338.383} C_VEL
LIN {X 0,Y 497.585,Z 261.329,A -85,B 0,C 180,E1 -6338.904,E2 -6338.904} C_VEL
LIN {X 0,Y 497.825,Z 249.464,A -85,B 0,C 180,E1 -6339.252,E2 -6339.252} C_VEL
LIN {X 0,Y 497.132,Z 243.713,A -85,B 0,C 180,E1 -6339.395,E2 -6339.395} C_VEL
LIN {X 0,Y 491.725,Z 225.031,A -85,B 0,C 180,E1 -6339.844,E2 -6339.844} C_VEL
LIN {X 0,Y 491.199,Z 219.224,A -85,B 0,C 180,E1 -6339.946,E2 -6339.946} C_VEL
LIN {X 0,Y 491.694,Z 151.546,A -85,B 0,C 180,E1 -6341.001,E2 -6341.001} C_VEL
LIN {X 0,Y 489.301,Z 140.042,A -85,B 0,C 180,E1 -6341.274,E2 -6341.274} C_VEL
LIN {X 0,Y 489.397,Z 132.091,A -85,B 0,C 180,E1 -6342.913,E2 -6342.913} C_VEL
LIN {X 0,Y 488.768,Z 127.605,A -85,B 0,C 180,E1 -6343.924,E2 -6343.924} C_VEL
LIN {X 0,Y 488.709,Z 127.609,A -85,B 0,C 180,E1 -6347.173,E2 -6347.173} C_VEL
LIN {X 0,Y 488.733,Z 127.61,A -85,B 0,C 180,E1 -6349.676,E2 -6349.676} C_VEL
LIN {X 0,Y 488.679,Z 127.609,A -85,B 0,C 180,E1 -6352.841,E2 -6352.841} C_VEL
LIN {X 0,Y 488.723,Z 127.607,A -85,B 0,C 180,E1 -6355.886,E2 -6355.886} C_VEL
LIN {X 0,Y 488.69,Z 127.608,A -85,B 0,C 180,E1 -6358.82,E2 -6358.82} C_VEL
LIN {X 0,Y 488.743,Z 127.605,A -85,B 0,C 180,E1 -6361.671,E2 -6361.671} C_VEL
LIN {X 0,Y 488.746,Z 127.6,A -85,B 0,C 180,E1 -6364.444,E2 -6364.444} C_VEL
LIN {X 0,Y 488.722,Z 127.609,A -85,B 0,C 180,E1 -6367.153,E2 -6367.153} C_VEL
LIN {X 0,Y 488.724,Z 127.604,A -85,B 0,C 180,E1 -6369.81,E2 -6369.81} C_VEL
LIN {X 0,Y 488.714,Z 127.604,A -85,B 0,C 180,E1 -6372.422,E2 -6372.422} C_VEL
LIN {X 0,Y 488.761,Z 127.605,A -85,B 0,C 180,E1 -6374.999,E2 -6374.999} C_VEL
LIN {X 0,Y 488.805,Z 127.593,A -85,B 0,C 180,E1 -6378.387,E2 -6378.387} C_VEL
LIN {X 0,Y 488.816,Z 127.592,A -85,B 0,C 180,E1 -6381.733,E2 -6381.733} C_VEL
LIN {X 0,Y 488.846,Z 127.588,A -85,B 0,C 180,E1 -6384.224,E2 -6384.224} C_VEL
LIN {X 0,Y 488.961,Z 127.574,A -85,B 0,C 180,E1 -6387.528,E2 -6387.528} C_VEL
LIN {X 0,Y 488.953,Z 127.582,A -85,B 0,C 180,E1 -6390.823,E2 -6390.823} C_VEL
LIN {X 0,Y 488.96,Z 127.578,A -85,B 0,C 180,E1 -6392.471,E2 -6392.471} C_VEL
LIN {X 0,Y 488.847,Z 127.587,A -85,B 0,C 180,E1 -6395.776,E2 -6395.776} C_VEL
LIN {X 0,Y 488.816,Z 127.595,A -85,B 0,C 180,E1 -6398.266,E2 -6398.266} C_VEL
LIN {X 0,Y 488.804,Z 127.593,A -85,B 0,C 180,E1 -6401.612,E2 -6401.612} C_VEL
LIN {X 0,Y 488.763,Z 127.6,A -85,B 0,C 180,E1 -6405,E2 -6405} C_VEL
LIN {X 0,Y 488.753,Z 127.607,A -85,B 0,C 180,E1 -6408.442,E2 -6408.442} C_VEL
LIN {X 0,Y 488.704,Z 127.606,A -85,B 0,C 180,E1 -6411.07,E2 -6411.07} C_VEL
LIN {X 0,Y 488.677,Z 127.61,A -85,B 0,C 180,E1 -6413.746,E2 -6413.746} C_VEL
LIN {X 0,Y 488.789,Z 127.595,A -85,B 0,C 180,E1 -6416.943,E2 -6416.943} C_VEL
LIN {X 0,Y 488.716,Z 127.609,A -85,B 0,C 180,E1 -6420.365,E2 -6420.365} C_VEL
LIN {X 0,Y 488.733,Z 127.603,A -85,B 0,C 180,E1 -6423.484,E2 -6423.484} C_VEL
LIN {X 0,Y 488.685,Z 127.611,A -85,B 0,C 180,E1 -6426.355,E2 -6426.355} C_VEL
LIN {X 0,Y 488.699,Z 127.606,A -85,B 0,C 180,E1 -6429.254,E2 -6429.254} C_VEL
LIN {X 0,Y 488.732,Z 127.603,A -85,B 0,C 180,E1 -6432.521,E2 -6432.521} C_VEL
LIN {X 0,Y 488.709,Z 127.606,A -85,B 0,C 180,E1 -6435.199,E2 -6435.199} C_VEL
LIN {X 0,Y 488.709,Z 127.606,A -85,B 0,C 180,E1 -6438.399,E2 -6438.399} C_VEL
LIN {X 0,Y 488.737,Z 127.601,A -85,B 0,C 180,E1 -6440.942,E2 -6440.942} C_VEL
LIN {X 0,Y 488.674,Z 127.614,A -85,B 0,C 180,E1 -6443.868,E2 -6443.868} C_VEL
LIN {X 0,Y 488.735,Z 127.602,A -85,B 0,C 180,E1 -6446.877,E2 -6446.877} C_VEL
LIN {X 0,Y 488.721,Z 127.608,A -85,B 0,C 180,E1 -6449.781,E2 -6449.781} C_VEL
LIN {X 0,Y 488.789,Z 127.598,A -85,B 0,C 180,E1 -6453.056,E2 -6453.056} C_VEL
LIN {X 0,Y 488.686,Z 127.607,A -85,B 0,C 180,E1 -6456.255,E2 -6456.255} C_VEL
LIN {X 0,Y 488.743,Z 127.607,A -85,B 0,C 180,E1 -6459.176,E2 -6459.176} C_VEL
LIN {X 0,Y 488.757,Z 127.602,A -85,B 0,C 180,E1 -6461.628,E2 -6461.628} C_VEL
LIN {X 0,Y 488.759,Z 127.604,A -85,B 0,C 180,E1 -6465,E2 -6465} C_VEL
LIN {X 0,Y 488.803,Z 127.593,A -85,B 0,C 180,E1 -6468.388,E2 -6468.388} C_VEL
LIN {X 0,Y 488.815,Z 127.592,A -85,B 0,C 180,E1 -6471.734,E2 -6471.734} C_VEL
LIN {X 0,Y 488.846,Z 127.588,A -85,B 0,C 180,E1 -6474.224,E2 -6474.224} C_VEL
LIN {X 0,Y 488.96,Z 127.575,A -85,B 0,C 180,E1 -6477.529,E2 -6477.529} C_VEL
LIN {X 0,Y 488.953,Z 127.582,A -85,B 0,C 180,E1 -6480.824,E2 -6480.824} C_VEL
LIN {X 0,Y 488.96,Z 127.577,A -85,B 0,C 180,E1 -6482.472,E2 -6482.472} C_VEL
LIN {X 0,Y 488.857,Z 127.586,A -85,B 0,C 180,E1 -6485.776,E2 -6485.776} C_VEL
LIN {X 0,Y 488.816,Z 127.594,A -85,B 0,C 180,E1 -6488.267,E2 -6488.267} C_VEL
LIN {X 0,Y 488.804,Z 127.593,A -85,B 0,C 180,E1 -6491.613,E2 -6491.613} C_VEL
LIN {X 0,Y 488.764,Z 127.6,A -85,B 0,C 180,E1 -6495.001,E2 -6495.001} C_VEL
LIN {X 0,Y 488.754,Z 127.607,A -85,B 0,C 180,E1 -6498.442,E2 -6498.442} C_VEL
LIN {X 0,Y 488.706,Z 127.606,A -85,B 0,C 180,E1 -6501.071,E2 -6501.071} C_VEL
LIN {X 0,Y 488.678,Z 127.61,A -85,B 0,C 180,E1 -6503.747,E2 -6503.747} C_VEL
LIN {X 0,Y 488.791,Z 127.595,A -85,B 0,C 180,E1 -6506.944,E2 -6506.944} C_VEL
LIN {X 0,Y 488.709,Z 127.611,A -85,B 0,C 180,E1 -6510.363,E2 -6510.363} C_VEL
LIN {X 0,Y 488.734,Z 127.602,A -85,B 0,C 180,E1 -6513.485,E2 -6513.485} C_VEL
LIN {X 0,Y 488.682,Z 127.613,A -85,B 0,C 180,E1 -6516.355,E2 -6516.355} C_VEL
LIN {X 0,Y 488.741,Z 127.601,A -85,B 0,C 180,E1 -6519.251,E2 -6519.251} C_VEL
LIN {X 0,Y 488.71,Z 127.608,A -85,B 0,C 180,E1 -6521.601,E2 -6521.601} C_VEL
LIN {X 0,Y 488.712,Z 127.604,A -85,B 0,C 180,E1 -6524.802,E2 -6524.802} C_VEL
LIN {X 0,Y 488.692,Z 127.61,A -85,B 0,C 180,E1 -6527.475,E2 -6527.475} C_VEL
LIN {X 0,Y 488.733,Z 127.608,A -85,B 0,C 180,E1 -6529.677,E2 -6529.677} C_VEL
LIN {X 0,Y 488.68,Z 127.608,A -85,B 0,C 180,E1 -6532.842,E2 -6532.842} C_VEL
LIN {X 0,Y 488.731,Z 127.607,A -85,B 0,C 180,E1 -6535.888,E2 -6535.888} C_VEL
LIN {X 0,Y 488.693,Z 127.608,A -85,B 0,C 180,E1 -6538.821,E2 -6538.821} C_VEL
LIN {X 0,Y 488.746,Z 127.607,A -85,B 0,C 180,E1 -6541.672,E2 -6541.672} C_VEL
LIN {X 0,Y 488.83,Z 127.697,A -85,B 0,C 180,E1 -6543.648,E2 -6543.648} C_VEL
LIN {X 0,Y 490.851,Z 138.253,A -85,B 0,C 180,E1 -6545.467,E2 -6545.467} C_VEL
LIN {X 0,Y 490.511,Z 150.731,A -85,B 0,C 180,E1 -6547.464,E2 -6547.464} C_VEL
LIN {X 0,Y 489.942,Z 165.943,A -85,B 0,C 180,E1 -6549.863,E2 -6549.863} C_VEL
LIN {X 0,Y 489.436,Z 182.501,A -85,B 0,C 180,E1 -6552.45,E2 -6552.45} C_VEL
LIN {X 0,Y 489.258,Z 191.134,A -85,B 0,C 180,E1 -6553.751,E2 -6553.751} C_VEL
LIN {X 0,Y 491.553,Z 208.023,A -85,B 0,C 180,E1 -6554.091,E2 -6554.091} C_VEL
LIN {X 0,Y 490.891,Z 300.459,A -85,B 0,C 180,E1 -6555.544,E2 -6555.544} C_VEL
LIN {X 0,Y 490.582,Z 312.534,A -85,B 0,C 180,E1 -6555.878,E2 -6555.878} C_VEL
LIN {X 0,Y 490.174,Z 324.713,A -85,B 0,C 180,E1 -6556.369,E2 -6556.369} C_VEL
LIN {X 0,Y 489.762,Z 337.065,A -85,B 0,C 180,E1 -6557.044,E2 -6557.044} C_VEL
LIN {X 0,Y 489.367,Z 348.452,A -85,B 0,C 180,E1 -6557.853,E2 -6557.853} C_VEL
LIN {X 0,Y 489.012,Z 359.246,A -85,B 0,C 180,E1 -6558.813,E2 -6558.813} C_VEL
LIN {X 0,Y 488.655,Z 368.704,A -85,B 0,C 180,E1 -6559.853,E2 -6559.853} C_VEL
LIN {X 0,Y 488.347,Z 377.841,A -85,B 0,C 180,E1 -6561.1,E2 -6561.1} C_VEL
LIN {X 0,Y 488.173,Z 385.207,A -85,B 0,C 180,E1 -6562.348,E2 -6562.348} C_VEL
LIN {X 0,Y 488.033,Z 390.867,A -85,B 0,C 180,E1 -6563.54,E2 -6563.54} C_VEL
LIN {X 0,Y 488.035,Z 395.012,A -85,B 0,C 180,E1 -6564.629,E2 -6564.629} C_VEL
LIN {X 0,Y 487.951,Z 398.696,A -85,B 0,C 180,E1 -6565.871,E2 -6565.871} C_VEL
LIN {X 0,Y 487.997,Z 400.599,A -85,B 0,C 180,E1 -6566.698,E2 -6566.698} C_VEL
LIN {X 0,Y 487.968,Z 402.023,A -85,B 0,C 180,E1 -6567.524,E2 -6567.524} C_VEL
LIN {X 0,Y 487.896,Z 403.027,A -85,B 0,C 180,E1 -6568.349,E2 -6568.349} C_VEL
LIN {X 0,Y 487.85,Z 403.634,A -85,B 0,C 180,E1 -6569.175,E2 -6569.175} C_VEL
LIN {X 0,Y 487.845,Z 403.843,A -85,B 0,C 180,E1 -6570,E2 -6570} C_VEL
LIN {X 0,Y 487.851,Z 403.607,A -85,B 0,C 180,E1 -6570.826,E2 -6570.826} C_VEL
LIN {X 0,Y 487.896,Z 402.97,A -85,B 0,C 180,E1 -6571.651,E2 -6571.651} C_VEL
LIN {X 0,Y 487.968,Z 401.936,A -85,B 0,C 180,E1 -6572.477,E2 -6572.477} C_VEL
LIN {X 0,Y 487.998,Z 400.485,A -85,B 0,C 180,E1 -6573.303,E2 -6573.303} C_VEL
LIN {X 0,Y 487.922,Z 397.443,A -85,B 0,C 180,E1 -6574.544,E2 -6574.544} C_VEL
LIN {X 0,Y 488.002,Z 393.339,A -85,B 0,C 180,E1 -6575.786,E2 -6575.786} C_VEL
LIN {X 0,Y 488.115,Z 387.025,A -85,B 0,C 180,E1 -6577.238,E2 -6577.238} C_VEL
LIN {X 0,Y 488.291,Z 380.145,A -85,B 0,C 180,E1 -6578.484,E2 -6578.484} C_VEL
LIN {X 0,Y 488.515,Z 371.602,A -85,B 0,C 180,E1 -6579.732,E2 -6579.732} C_VEL
LIN {X 0,Y 488.842,Z 362.804,A -85,B 0,C 180,E1 -6580.772,E2 -6580.772} C_VEL
LIN {X 0,Y 489.183,Z 352.18,A -85,B 0,C 180,E1 -6581.796,E2 -6581.796} C_VEL
LIN {X 0,Y 489.528,Z 341.518,A -85,B 0,C 180,E1 -6582.626,E2 -6582.626} C_VEL
LIN {X 0,Y 490.011,Z 329.258,A -85,B 0,C 180,E1 -6583.372,E2 -6583.372} C_VEL
LIN {X 0,Y 490.404,Z 316.864,A -85,B 0,C 180,E1 -6583.942,E2 -6583.942} C_VEL
LIN {X 0,Y 490.697,Z 304.241,A -85,B 0,C 180,E1 -6584.357,E2 -6584.357} C_VEL
LIN {X 0,Y 490.945,Z 289.678,A -85,B 0,C 180,E1 -6584.641,E2 -6584.641} C_VEL
LIN {X 0,Y 491.478,Z 206.773,A -85,B 0,C 180,E1 -6585.941,E2 -6585.941} C_VEL
LIN {X 0,Y 489.184,Z 189.423,A -85,B 0,C 180,E1 -6586.324,E2 -6586.324} C_VEL
LIN {X 0,Y 489.7,Z 168.672,A -85,B 0,C 180,E1 -6589.492,E2 -6589.492} C_VEL
LIN {X 0,Y 490.136,Z 151.724,A -85,B 0,C 180,E1 -6592.111,E2 -6592.111} C_VEL
LIN {X 0,Y 490.603,Z 137.542,A -85,B 0,C 180,E1 -6594.321,E2 -6594.321} C_VEL
LIN {X 0,Y 488.776,Z 127.604,A -85,B 0,C 180,E1 -6596.012,E2 -6596.012} C_VEL
LIN {X 0,Y 488.727,Z 127.61,A -85,B 0,C 180,E1 -6599.27,E2 -6599.27} C_VEL
LIN {X 0,Y 488.707,Z 127.614,A -85,B 0,C 180,E1 -6602.147,E2 -6602.147} C_VEL
LIN {X 0,Y 488.721,Z 127.606,A -85,B 0,C 180,E1 -6605.115,E2 -6605.115} C_VEL
LIN {X 0,Y 488.684,Z 127.615,A -85,B 0,C 180,E1 -6608.2,E2 -6608.2} C_VEL
LIN {X 0,Y 488.722,Z 127.609,A -85,B 0,C 180,E1 -6610.345,E2 -6610.345} C_VEL
LIN {X 0,Y 488.691,Z 127.613,A -85,B 0,C 180,E1 -6613.654,E2 -6613.654} C_VEL
LIN {X 0,Y 488.691,Z 127.609,A -85,B 0,C 180,E1 -6616.346,E2 -6616.346} C_VEL
LIN {X 0,Y 488.737,Z 127.607,A -85,B 0,C 180,E1 -6619.677,E2 -6619.677} C_VEL
LIN {X 0,Y 488.682,Z 127.607,A -85,B 0,C 180,E1 -6622.841,E2 -6622.841} C_VEL
LIN {X 0,Y 488.727,Z 127.605,A -85,B 0,C 180,E1 -6625.887,E2 -6625.887} C_VEL
LIN {X 0,Y 488.694,Z 127.606,A -85,B 0,C 180,E1 -6628.82,E2 -6628.82} C_VEL
LIN {X 0,Y 488.747,Z 127.605,A -85,B 0,C 180,E1 -6631.671,E2 -6631.671} C_VEL
LIN {X 0,Y 488.742,Z 127.599,A -85,B 0,C 180,E1 -6634.444,E2 -6634.444} C_VEL
LIN {X 0,Y 488.726,Z 127.608,A -85,B 0,C 180,E1 -6637.153,E2 -6637.153} C_VEL
LIN {X 0,Y 488.727,Z 127.603,A -85,B 0,C 180,E1 -6639.81,E2 -6639.81} C_VEL
LIN {X 0,Y 488.712,Z 127.604,A -85,B 0,C 180,E1 -6642.422,E2 -6642.422} C_VEL
LIN {X 0,Y 488.763,Z 127.605,A -85,B 0,C 180,E1 -6644.999,E2 -6644.999} C_VEL
LIN {X 0,Y 488.808,Z 127.597,A -85,B 0,C 180,E1 -6648.387,E2 -6648.387} C_VEL
LIN {X 0,Y 488.788,Z 127.598,A -85,B 0,C 180,E1 -6651.733,E2 -6651.733} C_VEL
LIN {X 0,Y 488.843,Z 127.594,A -85,B 0,C 180,E1 -6654.224,E2 -6654.224} C_VEL
LIN {X 0,Y 488.956,Z 127.578,A -85,B 0,C 180,E1 -6657.528,E2 -6657.528} C_VEL
LIN {X 0,Y 488.915,Z 127.586,A -85,B 0,C 180,E1 -6660.823,E2 -6660.823} C_VEL
LIN {X 0,Y 488.953,Z 127.583,A -85,B 0,C 180,E1 -6662.471,E2 -6662.471} C_VEL
LIN {X 0,Y 488.868,Z 127.792,A -85,B 0,C 180,E1 -6666.189,E2 -6666.189} C_VEL
LIN {X 0,Y 489.538,Z 132.902,A -85,B 0,C 180,E1 -6667.216,E2 -6667.216} C_VEL
LIN {X 0,Y 489.486,Z 140.888,A -85,B 0,C 180,E1 -6668.764,E2 -6668.764} C_VEL
LIN {X 0,Y 491.932,Z 153.057,A -85,B 0,C 180,E1 -6669.069,E2 -6669.069} C_VEL
LIN {X 0,Y 491.023,Z 248.478,A -85,B 0,C 180,E1 -6670.593,E2 -6670.593} C_VEL
LIN {X 0,Y 490.808,Z 262.138,A -85,B 0,C 180,E1 -6670.989,E2 -6670.989} C_VEL
LIN {X 0,Y 490.561,Z 274.482,A -85,B 0,C 180,E1 -6671.518,E2 -6671.518} C_VEL
LIN {X 0,Y 490.172,Z 286.453,A -85,B 0,C 180,E1 -6672.209,E2 -6672.209} C_VEL
LIN {X 0,Y 489.824,Z 297.353,A -85,B 0,C 180,E1 -6673.014,E2 -6673.014} C_VEL
LIN {X 0,Y 489.479,Z 307.209,A -85,B 0,C 180,E1 -6673.916,E2 -6673.916} C_VEL
LIN {X 0,Y 489.118,Z 316.688,A -85,B 0,C 180,E1 -6674.989,E2 -6674.989} C_VEL
LIN {X 0,Y 488.749,Z 325.896,A -85,B 0,C 180,E1 -6676.284,E2 -6676.284} C_VEL
LIN {X 0,Y 488.475,Z 333.232,A -85,B 0,C 180,E1 -6677.586,E2 -6677.586} C_VEL
LIN {X 0,Y 488.323,Z 339.027,A -85,B 0,C 180,E1 -6678.894,E2 -6678.894} C_VEL
LIN {X 0,Y 488.147,Z 343.556,A -85,B 0,C 180,E1 -6680.214,E2 -6680.214} C_VEL
LIN {X 0,Y 488.071,Z 345.934,A -85,B 0,C 180,E1 -6681.099,E2 -6681.099} C_VEL
LIN {X 0,Y 487.953,Z 347.772,A -85,B 0,C 180,E1 -6681.992,E2 -6681.992} C_VEL
LIN {X 0,Y 487.922,Z 349.136,A -85,B 0,C 180,E1 -6682.886,E2 -6682.886} C_VEL
LIN {X 0,Y 487.858,Z 350.04,A -85,B 0,C 180,E1 -6683.788,E2 -6683.788} C_VEL
LIN {X 0,Y 487.834,Z 350.446,A -85,B 0,C 180,E1 -6684.822,E2 -6684.822} C_VEL
LIN {X 0,Y 487.892,Z 350.358,A -85,B 0,C 180,E1 -6685.603,E2 -6685.603} C_VEL
LIN {X 0,Y 487.945,Z 349.553,A -85,B 0,C 180,E1 -6686.747,E2 -6686.747} C_VEL
LIN {X 0,Y 487.976,Z 347.1,A -85,B 0,C 180,E1 -6688.377,E2 -6688.377} C_VEL
LIN {X 0,Y 488.132,Z 343.622,A -85,B 0,C 180,E1 -6689.777,E2 -6689.777} C_VEL
LIN {X 0,Y 488.208,Z 338.674,A -85,B 0,C 180,E1 -6691.214,E2 -6691.214} C_VEL
LIN {X 0,Y 488.514,Z 332.134,A -85,B 0,C 180,E1 -6692.649,E2 -6692.649} C_VEL
LIN {X 0,Y 488.761,Z 324.675,A -85,B 0,C 180,E1 -6693.926,E2 -6693.926} C_VEL
LIN {X 0,Y 489.102,Z 315.337,A -85,B 0,C 180,E1 -6695.209,E2 -6695.209} C_VEL
LIN {X 0,Y 489.421,Z 305.521,A -85,B 0,C 180,E1 -6696.283,E2 -6696.283} C_VEL
LIN {X 0,Y 489.826,Z 295.328,A -85,B 0,C 180,E1 -6697.186,E2 -6697.186} C_VEL
LIN {X 0,Y 490.18,Z 284.68,A -85,B 0,C 180,E1 -6697.948,E2 -6697.948} C_VEL
LIN {X 0,Y 490.501,Z 272.649,A -85,B 0,C 180,E1 -6698.621,E2 -6698.621} C_VEL
LIN {X 0,Y 490.728,Z 259.402,A -85,B 0,C 180,E1 -6699.163,E2 -6699.163} C_VEL
LIN {X 0,Y 490.97,Z 246.945,A -85,B 0,C 180,E1 -6699.505,E2 -6699.505} C_VEL
LIN {X 0,Y 491.199,Z 219.224,A -85,B 0,C 180,E1 -6699.946,E2 -6699.946} C_VEL
LIN {X 0,Y 490.658,Z 213.417,A -85,B 0,C 180,E1 -6700.053,E2 -6700.053} C_VEL
LIN {X 0,Y 485.253,Z 194.73,A -85,B 0,C 180,E1 -6700.514,E2 -6700.514} C_VEL
LIN {X 0,Y 484.629,Z 188.924,A -85,B 0,C 180,E1 -6700.626,E2 -6700.626} C_VEL
LIN {X 0,Y 484.773,Z 152.262,A -85,B 0,C 180,E1 -6701.216,E2 -6701.216} C_VEL
LIN {X 0,Y 482.342,Z 140.399,A -85,B 0,C 180,E1 -6701.494,E2 -6701.494} C_VEL
LIN {X 0,Y 482.303,Z 132.063,A -85,B 0,C 180,E1 -6703.232,E2 -6703.232} C_VEL
LIN {X 0,Y 481.72,Z 128.483,A -85,B 0,C 180,E1 -6704.029,E2 -6704.029} C_VEL
LIN {X 0,Y 481.644,Z 128.487,A -85,B 0,C 180,E1 -6706.851,E2 -6706.851} C_VEL
LIN {X 0,Y 481.676,Z 128.484,A -85,B 0,C 180,E1 -6710.059,E2 -6710.059} C_VEL
LIN {X 0,Y 481.625,Z 128.491,A -85,B 0,C 180,E1 -6713.253,E2 -6713.253} C_VEL
LIN {X 0,Y 481.676,Z 128.481,A -85,B 0,C 180,E1 -6716.327,E2 -6716.327} C_VEL
LIN {X 0,Y 481.649,Z 128.492,A -85,B 0,C 180,E1 -6719.417,E2 -6719.417} C_VEL
LIN {X 0,Y 481.699,Z 128.478,A -85,B 0,C 180,E1 -6722.168,E2 -6722.168} C_VEL
LIN {X 0,Y 481.717,Z 128.479,A -85,B 0,C 180,E1 -6724.97,E2 -6724.97} C_VEL
LIN {X 0,Y 481.648,Z 128.487,A -85,B 0,C 180,E1 -6727.704,E2 -6727.704} C_VEL
LIN {X 0,Y 481.703,Z 128.477,A -85,B 0,C 180,E1 -6730.393,E2 -6730.393} C_VEL
LIN {X 0,Y 481.678,Z 128.487,A -85,B 0,C 180,E1 -6733.033,E2 -6733.033} C_VEL
LIN {X 0,Y 481.689,Z 128.481,A -85,B 0,C 180,E1 -6735.638,E2 -6735.638} C_VEL
LIN {X 0,Y 481.75,Z 128.472,A -85,B 0,C 180,E1 -6738.215,E2 -6738.215} C_VEL
LIN {X 0,Y 481.762,Z 128.471,A -85,B 0,C 180,E1 -6741.611,E2 -6741.611} C_VEL
LIN {X 0,Y 481.807,Z 128.465,A -85,B 0,C 180,E1 -6744.139,E2 -6744.139} C_VEL
LIN {X 0,Y 481.927,Z 128.451,A -85,B 0,C 180,E1 -6747.492,E2 -6747.492} C_VEL
LIN {X 0,Y 481.904,Z 128.46,A -85,B 0,C 180,E1 -6750.835,E2 -6750.835} C_VEL
LIN {X 0,Y 481.927,Z 128.454,A -85,B 0,C 180,E1 -6752.507,E2 -6752.507} C_VEL
LIN {X 0,Y 481.807,Z 128.464,A -85,B 0,C 180,E1 -6755.86,E2 -6755.86} C_VEL
LIN {X 0,Y 481.762,Z 128.475,A -85,B 0,C 180,E1 -6758.388,E2 -6758.388} C_VEL
LIN {X 0,Y 481.749,Z 128.472,A -85,B 0,C 180,E1 -6761.785,E2 -6761.785} C_VEL
LIN {X 0,Y 481.742,Z 128.473,A -85,B 0,C 180,E1 -6765.224,E2 -6765.224} C_VEL
LIN {X 0,Y 481.71,Z 128.48,A -85,B 0,C 180,E1 -6768.721,E2 -6768.721} C_VEL
LIN {X 0,Y 481.643,Z 128.485,A -85,B 0,C 180,E1 -6771.394,E2 -6771.394} C_VEL
LIN {X 0,Y 481.658,Z 128.489,A -85,B 0,C 180,E1 -6774.114,E2 -6774.114} C_VEL
LIN {X 0,Y 481.744,Z 128.472,A -85,B 0,C 180,E1 -6777.139,E2 -6777.139} C_VEL
LIN {X 0,Y 481.685,Z 128.482,A -85,B 0,C 180,E1 -6779.74,E2 -6779.74} C_VEL
LIN {X 0,Y 481.671,Z 128.483,A -85,B 0,C 180,E1 -6782.674,E2 -6782.674} C_VEL
LIN {X 0,Y 481.639,Z 128.489,A -85,B 0,C 180,E1 -6785.709,E2 -6785.709} C_VEL
LIN {X 0,Y 481.668,Z 128.482,A -85,B 0,C 180,E1 -6788.859,E2 -6788.859} C_VEL
LIN {X 0,Y 481.671,Z 128.486,A -85,B 0,C 180,E1 -6792.158,E2 -6792.158} C_VEL
LIN {X 0,Y 481.657,Z 128.484,A -85,B 0,C 180,E1 -6794.457,E2 -6794.457} C_VEL
LIN {X 0,Y 481.645,Z 128.492,A -85,B 0,C 180,E1 -6797.839,E2 -6797.839} C_VEL
LIN {X 0,Y 481.711,Z 128.476,A -85,B 0,C 180,E1 -6800.646,E2 -6800.646} C_VEL
LIN {X 0,Y 481.633,Z 128.487,A -85,B 0,C 180,E1 -6804.291,E2 -6804.291} C_VEL
LIN {X 0,Y 481.67,Z 128.486,A -85,B 0,C 180,E1 -6807.326,E2 -6807.326} C_VEL
LIN {X 0,Y 481.676,Z 128.481,A -85,B 0,C 180,E1 -6810.259,E2 -6810.259} C_VEL
LIN {X 0,Y 481.743,Z 128.476,A -85,B 0,C 180,E1 -6813.112,E2 -6813.112} C_VEL
LIN {X 0,Y 481.671,Z 128.483,A -85,B 0,C 180,E1 -6815.887,E2 -6815.887} C_VEL
LIN {X 0,Y 481.699,Z 128.482,A -85,B 0,C 180,E1 -6819.028,E2 -6819.028} C_VEL
LIN {X 0,Y 481.704,Z 128.477,A -85,B 0,C 180,E1 -6822.159,E2 -6822.159} C_VEL
LIN {X 0,Y 481.74,Z 128.476,A -85,B 0,C 180,E1 -6824.776,E2 -6824.776} C_VEL
LIN {X 0,Y 481.748,Z 128.472,A -85,B 0,C 180,E1 -6828.215,E2 -6828.215} C_VEL
LIN {X 0,Y 481.76,Z 128.472,A -85,B 0,C 180,E1 -6831.612,E2 -6831.612} C_VEL
LIN {X 0,Y 481.806,Z 128.465,A -85,B 0,C 180,E1 -6834.14,E2 -6834.14} C_VEL
LIN {X 0,Y 481.927,Z 128.451,A -85,B 0,C 180,E1 -6837.493,E2 -6837.493} C_VEL
LIN {X 0,Y 481.904,Z 128.461,A -85,B 0,C 180,E1 -6840.836,E2 -6840.836} C_VEL
LIN {X 0,Y 481.927,Z 128.454,A -85,B 0,C 180,E1 -6842.508,E2 -6842.508} C_VEL
LIN {X 0,Y 481.817,Z 128.463,A -85,B 0,C 180,E1 -6845.861,E2 -6845.861} C_VEL
LIN {X 0,Y 481.762,Z 128.474,A -85,B 0,C 180,E1 -6848.389,E2 -6848.389} C_VEL
LIN {X 0,Y 481.75,Z 128.472,A -85,B 0,C 180,E1 -6851.785,E2 -6851.785} C_VEL
LIN {X 0,Y 481.743,Z 128.473,A -85,B 0,C 180,E1 -6855.224,E2 -6855.224} C_VEL
LIN {X 0,Y 481.711,Z 128.481,A -85,B 0,C 180,E1 -6858.722,E2 -6858.722} C_VEL
LIN {X 0,Y 481.644,Z 128.485,A -85,B 0,C 180,E1 -6861.395,E2 -6861.395} C_VEL
LIN {X 0,Y 481.66,Z 128.488,A -85,B 0,C 180,E1 -6864.114,E2 -6864.114} C_VEL
LIN {X 0,Y 481.746,Z 128.472,A -85,B 0,C 180,E1 -6867.14,E2 -6867.14} C_VEL
LIN {X 0,Y 481.678,Z 128.483,A -85,B 0,C 180,E1 -6869.741,E2 -6869.741} C_VEL
LIN {X 0,Y 481.671,Z 128.483,A -85,B 0,C 180,E1 -6872.675,E2 -6872.675} C_VEL
LIN {X 0,Y 481.636,Z 128.489,A -85,B 0,C 180,E1 -6875.71,E2 -6875.71} C_VEL
LIN {X 0,Y 481.713,Z 128.477,A -85,B 0,C 180,E1 -6879.354,E2 -6879.354} C_VEL
LIN {X 0,Y 481.648,Z 128.49,A -85,B 0,C 180,E1 -6882.161,E2 -6882.161} C_VEL
LIN {X 0,Y 481.66,Z 128.486,A -85,B 0,C 180,E1 -6885.543,E2 -6885.543} C_VEL
LIN {X 0,Y 481.657,Z 128.483,A -85,B 0,C 180,E1 -6888.959,E2 -6888.959} C_VEL
LIN {X 0,Y 481.656,Z 128.488,A -85,B 0,C 180,E1 -6891.993,E2 -6891.993} C_VEL
LIN {X 0,Y 481.689,Z 128.482,A -85,B 0,C 180,E1 -6895.318,E2 -6895.318} C_VEL
LIN {X 0,Y 481.646,Z 128.487,A -85,B 0,C 180,E1 -6898.312,E2 -6898.312} C_VEL
LIN {X 0,Y 481.701,Z 128.483,A -85,B 0,C 180,E1 -6901.219,E2 -6901.219} C_VEL
LIN {X 0,Y 481.781,Z 128.666,A -85,B 0,C 180,E1 -6903.465,E2 -6903.465} C_VEL
LIN {X 0,Y 484.028,Z 140.634,A -85,B 0,C 180,E1 -6905.556,E2 -6905.556} C_VEL
LIN {X 0,Y 483.289,Z 160.022,A -85,B 0,C 180,E1 -6908.682,E2 -6908.682} C_VEL
LIN {X 0,Y 482.62,Z 179.352,A -85,B 0,C 180,E1 -6911.755,E2 -6911.755} C_VEL
LIN {X 0,Y 482.23,Z 190.513,A -85,B 0,C 180,E1 -6913.512,E2 -6913.512} C_VEL
LIN {X 0,Y 484.686,Z 208.791,A -85,B 0,C 180,E1 -6913.889,E2 -6913.889} C_VEL
LIN {X 0,Y 483.998,Z 299.358,A -85,B 0,C 180,E1 -6915.333,E2 -6915.333} C_VEL
LIN {X 0,Y 483.641,Z 312.412,A -85,B 0,C 180,E1 -6915.698,E2 -6915.698} C_VEL
LIN {X 0,Y 483.212,Z 325.086,A -85,B 0,C 180,E1 -6916.222,E2 -6916.222} C_VEL
LIN {X 0,Y 482.805,Z 336.415,A -85,B 0,C 180,E1 -6916.854,E2 -6916.854} C_VEL
LIN {X 0,Y 482.349,Z 348.645,A -85,B 0,C 180,E1 -6917.738,E2 -6917.738} C_VEL
LIN {X 0,Y 481.964,Z 359.76,A -85,B 0,C 180,E1 -6918.754,E2 -6918.754} C_VEL
LIN {X 0,Y 481.521,Z 369.851,A -85,B 0,C 180,E1 -6919.913,E2 -6919.913} C_VEL
LIN {X 0,Y 481.237,Z 378.744,A -85,B 0,C 180,E1 -6921.18,E2 -6921.18} C_VEL
LIN {X 0,Y 481.05,Z 385.837,A -85,B 0,C 180,E1 -6922.445,E2 -6922.445} C_VEL
LIN {X 0,Y 480.892,Z 392.099,A -85,B 0,C 180,E1 -6923.861,E2 -6923.861} C_VEL
LIN {X 0,Y 480.899,Z 395.951,A -85,B 0,C 180,E1 -6924.97,E2 -6924.97} C_VEL
LIN {X 0,Y 480.848,Z 398.292,A -85,B 0,C 180,E1 -6925.809,E2 -6925.809} C_VEL
LIN {X 0,Y 480.919,Z 400.202,A -85,B 0,C 180,E1 -6926.649,E2 -6926.649} C_VEL
LIN {X 0,Y 480.879,Z 401.631,A -85,B 0,C 180,E1 -6927.487,E2 -6927.487} C_VEL
LIN {X 0,Y 480.827,Z 402.638,A -85,B 0,C 180,E1 -6928.325,E2 -6928.325} C_VEL
LIN {X 0,Y 480.775,Z 403.246,A -85,B 0,C 180,E1 -6929.163,E2 -6929.163} C_VEL
LIN {X 0,Y 480.768,Z 403.455,A -85,B 0,C 180,E1 -6930,E2 -6930} C_VEL
LIN {X 0,Y 480.776,Z 403.219,A -85,B 0,C 180,E1 -6930.838,E2 -6930.838} C_VEL
LIN {X 0,Y 480.828,Z 402.58,A -85,B 0,C 180,E1 -6931.675,E2 -6931.675} C_VEL
LIN {X 0,Y 480.879,Z 401.543,A -85,B 0,C 180,E1 -6932.513,E2 -6932.513} C_VEL
LIN {X 0,Y 480.919,Z 400.089,A -85,B 0,C 180,E1 -6933.351,E2 -6933.351} C_VEL
LIN {X 0,Y 480.84,Z 397.041,A -85,B 0,C 180,E1 -6934.611,E2 -6934.611} C_VEL
LIN {X 0,Y 480.899,Z 392.928,A -85,B 0,C 180,E1 -6935.872,E2 -6935.872} C_VEL
LIN {X 0,Y 481.034,Z 386.603,A -85,B 0,C 180,E1 -6937.345,E2 -6937.345} C_VEL
LIN {X 0,Y 481.214,Z 379.707,A -85,B 0,C 180,E1 -6938.61,E2 -6938.61} C_VEL
LIN {X 0,Y 481.471,Z 371.151,A -85,B 0,C 180,E1 -6939.876,E2 -6939.876} C_VEL
LIN {X 0,Y 481.803,Z 362.344,A -85,B 0,C 180,E1 -6940.931,E2 -6940.931} C_VEL
LIN {X 0,Y 482.174,Z 351.958,A -85,B 0,C 180,E1 -6941.948,E2 -6941.948} C_VEL
LIN {X 0,Y 482.583,Z 340.76,A -85,B 0,C 180,E1 -6942.832,E2 -6942.832} C_VEL
LIN {X 0,Y 483.08,Z 328.783,A -85,B 0,C 180,E1 -6943.568,E2 -6943.568} C_VEL
LIN {X 0,Y 483.509,Z 316.379,A -85,B 0,C 180,E1 -6944.145,E2 -6944.145} C_VEL
LIN {X 0,Y 483.829,Z 303.746,A -85,B 0,C 180,E1 -6944.565,E2 -6944.565} C_VEL
LIN {X 0,Y 484.09,Z 289.211,A -85,B 0,C 180,E1 -6944.853,E2 -6944.853} C_VEL
LIN {X 0,Y 484.608,Z 206.99,A -85,B 0,C 180,E1 -6946.173,E2 -6946.173} C_VEL
LIN {X 0,Y 482.2,Z 189.08,A -85,B 0,C 180,E1 -6946.567,E2 -6946.567} C_VEL
LIN {X 0,Y 482.726,Z 168.321,A -85,B 0,C 180,E1 -6949.786,E2 -6949.786} C_VEL
LIN {X 0,Y 483.224,Z 151.369,A -85,B 0,C 180,E1 -6952.444,E2 -6952.444} C_VEL
LIN {X 0,Y 483.659,Z 138.604,A -85,B 0,C 180,E1 -6954.465,E2 -6954.465} C_VEL
LIN {X 0,Y 481.74,Z 128.48,A -85,B 0,C 180,E1 -6956.246,E2 -6956.246} C_VEL
LIN {X 0,Y 481.682,Z 128.49,A -85,B 0,C 180,E1 -6958.903,E2 -6958.903} C_VEL
LIN {X 0,Y 481.661,Z 128.492,A -85,B 0,C 180,E1 -6962.189,E2 -6962.189} C_VEL
LIN {X 0,Y 481.692,Z 128.484,A -85,B 0,C 180,E1 -6964.682,E2 -6964.682} C_VEL
LIN {X 0,Y 481.658,Z 128.492,A -85,B 0,C 180,E1 -6968.007,E2 -6968.007} C_VEL
LIN {X 0,Y 481.66,Z 128.485,A -85,B 0,C 180,E1 -6971.042,E2 -6971.042} C_VEL
LIN {X 0,Y 481.663,Z 128.486,A -85,B 0,C 180,E1 -6974.457,E2 -6974.457} C_VEL
LIN {X 0,Y 481.651,Z 128.489,A -85,B 0,C 180,E1 -6977.839,E2 -6977.839} C_VEL
LIN {X 0,Y 481.664,Z 128.48,A -85,B 0,C 180,E1 -6980.654,E2 -6980.654} C_VEL
LIN {X 0,Y 481.631,Z 128.49,A -85,B 0,C 180,E1 -6983.376,E2 -6983.376} C_VEL
LIN {X 0,Y 481.68,Z 128.479,A -85,B 0,C 180,E1 -6986.327,E2 -6986.327} C_VEL
LIN {X 0,Y 481.653,Z 128.489,A -85,B 0,C 180,E1 -6989.417,E2 -6989.417} C_VEL
LIN {X 0,Y 481.703,Z 128.479,A -85,B 0,C 180,E1 -6992.168,E2 -6992.168} C_VEL
LIN {X 0,Y 481.715,Z 128.478,A -85,B 0,C 180,E1 -6994.969,E2 -6994.969} C_VEL
LIN {X 0,Y 481.652,Z 128.487,A -85,B 0,C 180,E1 -6997.705,E2 -6997.705} C_VEL
LIN {X 0,Y 481.706,Z 128.478,A -85,B 0,C 180,E1 -7000.393,E2 -7000.393} C_VEL
LIN {X 0,Y 481.677,Z 128.488,A -85,B 0,C 180,E1 -7003.033,E2 -7003.033} C_VEL
LIN {X 0,Y 481.689,Z 128.481,A -85,B 0,C 180,E1 -7005.638,E2 -7005.638} C_VEL
LIN {X 0,Y 481.754,Z 128.474,A -85,B 0,C 180,E1 -7008.215,E2 -7008.215} C_VEL
LIN {X 0,Y 481.742,Z 128.476,A -85,B 0,C 180,E1 -7011.611,E2 -7011.611} C_VEL
LIN {X 0,Y 481.802,Z 128.471,A -85,B 0,C 180,E1 -7014.139,E2 -7014.139} C_VEL
LIN {X 0,Y 481.923,Z 128.454,A -85,B 0,C 180,E1 -7017.492,E2 -7017.492} C_VEL
LIN {X 0,Y 481.942,Z 128.452,A -85,B 0,C 180,E1 -7020,E2 -7020} C_VEL
LIN {X 0,Y 481.919,Z 128.46,A -85,B 0,C 180,E1 -7022.507,E2 -7022.507} C_VEL
LIN {X 0,Y 481.803,Z 128.54,A -85,B 0,C 180,E1 -7025.965,E2 -7025.965} C_VEL
LIN {X 0,Y 482.625,Z 134.153,A -85,B 0,C 180,E1 -7027.11,E2 -7027.11} C_VEL
LIN {X 0,Y 482.539,Z 141.311,A -85,B 0,C 180,E1 -7028.506,E2 -7028.506} C_VEL
LIN {X 0,Y 485.143,Z 153.634,A -85,B 0,C 180,E1 -7028.827,E2 -7028.827} C_VEL
LIN {X 0,Y 484.173,Z 248.536,A -85,B 0,C 180,E1 -7030.374,E2 -7030.374} C_VEL
LIN {X 0,Y 483.968,Z 262.246,A -85,B 0,C 180,E1 -7030.775,E2 -7030.775} C_VEL
LIN {X 0,Y 483.676,Z 274.703,A -85,B 0,C 180,E1 -7031.312,E2 -7031.312} C_VEL
LIN {X 0,Y 483.306,Z 285.892,A -85,B 0,C 180,E1 -7031.959,E2 -7031.959} C_VEL
LIN {X 0,Y 482.911,Z 297.482,A -85,B 0,C 180,E1 -7032.818,E2 -7032.818} C_VEL
LIN {X 0,Y 482.51,Z 308.044,A -85,B 0,C 180,E1 -7033.798,E2 -7033.798} C_VEL
LIN {X 0,Y 482.166,Z 316.6,A -85,B 0,C 180,E1 -7034.778,E2 -7034.778} C_VEL
LIN {X 0,Y 481.853,Z 324.137,A -85,B 0,C 180,E1 -7035.818,E2 -7035.818} C_VEL
LIN {X 0,Y 481.497,Z 332.184,A -85,B 0,C 180,E1 -7037.191,E2 -7037.191} C_VEL
LIN {X 0,Y 481.294,Z 337.607,A -85,B 0,C 180,E1 -7038.35,E2 -7038.35} C_VEL
LIN {X 0,Y 481.154,Z 342.38,A -85,B 0,C 180,E1 -7039.63,E2 -7039.63} C_VEL
LIN {X 0,Y 481.018,Z 345.625,A -85,B 0,C 180,E1 -7040.758,E2 -7040.758} C_VEL
LIN {X 0,Y 480.863,Z 348.832,A -85,B 0,C 180,E1 -7042.333,E2 -7042.333} C_VEL
LIN {X 0,Y 480.812,Z 349.97,A -85,B 0,C 180,E1 -7043.244,E2 -7043.244} C_VEL
LIN {X 0,Y 480.754,Z 350.65,A -85,B 0,C 180,E1 -7044.162,E2 -7044.162} C_VEL
LIN {X 0,Y 480.782,Z 350.863,A -85,B 0,C 180,E1 -7045.082,E2 -7045.082} C_VEL
LIN {X 0,Y 480.803,Z 350.544,A -85,B 0,C 180,E1 -7046.009,E2 -7046.009} C_VEL
LIN {X 0,Y 480.854,Z 349.763,A -85,B 0,C 180,E1 -7046.941,E2 -7046.941} C_VEL
LIN {X 0,Y 480.879,Z 348.442,A -85,B 0,C 180,E1 -7047.883,E2 -7047.883} C_VEL
LIN {X 0,Y 480.994,Z 345.436,A -85,B 0,C 180,E1 -7049.306,E2 -7049.306} C_VEL
LIN {X 0,Y 481.131,Z 341.076,A -85,B 0,C 180,E1 -7050.747,E2 -7050.747} C_VEL
LIN {X 0,Y 481.326,Z 335.517,A -85,B 0,C 180,E1 -7052.126,E2 -7052.126} C_VEL
LIN {X 0,Y 481.559,Z 328.767,A -85,B 0,C 180,E1 -7053.431,E2 -7053.431} C_VEL
LIN {X 0,Y 481.911,Z 320.821,A -85,B 0,C 180,E1 -7054.663,E2 -7054.663} C_VEL
LIN {X 0,Y 482.209,Z 311.924,A -85,B 0,C 180,E1 -7055.789,E2 -7055.789} C_VEL
LIN {X 0,Y 482.61,Z 302.251,A -85,B 0,C 180,E1 -7056.78,E2 -7056.78} C_VEL
LIN {X 0,Y 483.011,Z 291.49,A -85,B 0,C 180,E1 -7057.67,E2 -7057.67} C_VEL
LIN {X 0,Y 483.342,Z 280.403,A -85,B 0,C 180,E1 -7058.403,E2 -7058.403} C_VEL
LIN {X 0,Y 483.697,Z 268.744,A -85,B 0,C 180,E1 -7059,E2 -7059} C_VEL
LIN {X 0,Y 483.929,Z 256.217,A -85,B 0,C 180,E1 -7059.464,E2 -7059.464} C_VEL
LIN {X 0,Y 484.114,Z 242.736,A -85,B 0,C 180,E1 -7059.783,E2 -7059.783} C_VEL
LIN {X 0,Y 484.629,Z 188.924,A -85,B 0,C 180,E1 -7060.626,E2 -7060.626} C_VEL
LIN {X 0,Y 484.007,Z 183.12,A -85,B 0,C 180,E1 -7060.74,E2 -7060.74} C_VEL
LIN {X 0,Y 478.583,Z 164.462,A -85,B 0,C 180,E1 -7061.224,E2 -7061.224} C_VEL
LIN {X 0,Y 478.034,Z 158.659,A -85,B 0,C 180,E1 -7061.338,E2 -7061.338} C_VEL
LIN {X 0,Y 477.876,Z 152.828,A -85,B 0,C 180,E1 -7061.44,E2 -7061.44} C_VEL
LIN {X 0,Y 475.395,Z 140.648,A -85,B 0,C 180,E1 -7061.741,E2 -7061.741} C_VEL
LIN {X 0,Y 475.381,Z 133.674,A -85,B 0,C 180,E1 -7063.204,E2 -7063.204} C_VEL
LIN {X 0,Y 474.681,Z 129.359,A -85,B 0,C 180,E1 -7064.167,E2 -7064.167} C_VEL
LIN {X 0,Y 474.625,Z 129.367,A -85,B 0,C 180,E1 -7067.763,E2 -7067.763} C_VEL
LIN {X 0,Y 474.633,Z 129.358,A -85,B 0,C 180,E1 -7070.453,E2 -7070.453} C_VEL
LIN {X 0,Y 474.588,Z 129.371,A -85,B 0,C 180,E1 -7073.676,E2 -7073.676} C_VEL
LIN {X 0,Y 474.624,Z 129.36,A -85,B 0,C 180,E1 -7076.778,E2 -7076.778} C_VEL
LIN {X 0,Y 474.604,Z 129.366,A -85,B 0,C 180,E1 -7079.769,E2 -7079.769} C_VEL
LIN {X 0,Y 474.697,Z 129.351,A -85,B 0,C 180,E1 -7082.68,E2 -7082.68} C_VEL
LIN {X 0,Y 474.656,Z 129.361,A -85,B 0,C 180,E1 -7085.507,E2 -7085.507} C_VEL
LIN {X 0,Y 474.669,Z 129.361,A -85,B 0,C 180,E1 -7089.185,E2 -7089.185} C_VEL
LIN {X 0,Y 474.645,Z 129.357,A -85,B 0,C 180,E1 -7091.884,E2 -7091.884} C_VEL
LIN {X 0,Y 474.699,Z 129.351,A -85,B 0,C 180,E1 -7094.544,E2 -7094.544} C_VEL
LIN {X 0,Y 474.703,Z 129.349,A -85,B 0,C 180,E1 -7098.037,E2 -7098.037} C_VEL
LIN {X 0,Y 474.727,Z 129.349,A -85,B 0,C 180,E1 -7101.486,E2 -7101.486} C_VEL
LIN {X 0,Y 474.769,Z 129.341,A -85,B 0,C 180,E1 -7104.052,E2 -7104.052} C_VEL
LIN {X 0,Y 474.893,Z 129.327,A -85,B 0,C 180,E1 -7107.455,E2 -7107.455} C_VEL
LIN {X 0,Y 474.911,Z 129.324,A -85,B 0,C 180,E1 -7110,E2 -7110} C_VEL
LIN {X 0,Y 474.893,Z 129.331,A -85,B 0,C 180,E1 -7112.544,E2 -7112.544} C_VEL
LIN {X 0,Y 474.77,Z 129.342,A -85,B 0,C 180,E1 -7115.947,E2 -7115.947} C_VEL
LIN {X 0,Y 474.727,Z 129.353,A -85,B 0,C 180,E1 -7118.513,E2 -7118.513} C_VEL
LIN {X 0,Y 474.702,Z 129.351,A -85,B 0,C 180,E1 -7121.962,E2 -7121.962} C_VEL
LIN {X 0,Y 474.699,Z 129.35,A -85,B 0,C 180,E1 -7125.455,E2 -7125.455} C_VEL
LIN {X 0,Y 474.663,Z 129.356,A -85,B 0,C 180,E1 -7129.01,E2 -7129.01} C_VEL
LIN {X 0,Y 474.586,Z 129.365,A -85,B 0,C 180,E1 -7131.729,E2 -7131.729} C_VEL
LIN {X 0,Y 474.638,Z 129.363,A -85,B 0,C 180,E1 -7134.494,E2 -7134.494} C_VEL
LIN {X 0,Y 474.678,Z 129.352,A -85,B 0,C 180,E1 -7137.334,E2 -7137.334} C_VEL
LIN {X 0,Y 474.611,Z 129.368,A -85,B 0,C 180,E1 -7140.229,E2 -7140.229} C_VEL
LIN {X 0,Y 474.64,Z 129.357,A -85,B 0,C 180,E1 -7143.22,E2 -7143.22} C_VEL
LIN {X 0,Y 474.59,Z 129.368,A -85,B 0,C 180,E1 -7146.323,E2 -7146.323} C_VEL
LIN {X 0,Y 474.624,Z 129.363,A -85,B 0,C 180,E1 -7149.648,E2 -7149.648} C_VEL
LIN {X 0,Y 474.649,Z 129.356,A -85,B 0,C 180,E1 -7152.93,E2 -7152.93} C_VEL
LIN {X 0,Y 474.606,Z 129.369,A -85,B 0,C 180,E1 -7155.895,E2 -7155.895} C_VEL
LIN {X 0,Y 474.638,Z 129.358,A -85,B 0,C 180,E1 -7159.039,E2 -7159.039} C_VEL
LIN {X 0,Y 474.613,Z 129.369,A -85,B 0,C 180,E1 -7161.703,E2 -7161.703} C_VEL
LIN {X 0,Y 474.621,Z 129.36,A -85,B 0,C 180,E1 -7164.726,E2 -7164.726} C_VEL
LIN {X 0,Y 474.634,Z 129.363,A -85,B 0,C 180,E1 -7167.788,E2 -7167.788} C_VEL
LIN {X 0,Y 474.621,Z 129.361,A -85,B 0,C 180,E1 -7170.885,E2 -7170.885} C_VEL
LIN {X 0,Y 474.658,Z 129.361,A -85,B 0,C 180,E1 -7173.629,E2 -7173.629} C_VEL
LIN {X 0,Y 474.632,Z 129.359,A -85,B 0,C 180,E1 -7176.642,E2 -7176.642} C_VEL
LIN {X 0,Y 474.654,Z 129.356,A -85,B 0,C 180,E1 -7180.09,E2 -7180.09} C_VEL
LIN {X 0,Y 474.648,Z 129.359,A -85,B 0,C 180,E1 -7182.775,E2 -7182.775} C_VEL
LIN {X 0,Y 474.646,Z 129.361,A -85,B 0,C 180,E1 -7185.421,E2 -7185.421} C_VEL
LIN {X 0,Y 474.702,Z 129.349,A -85,B 0,C 180,E1 -7188.038,E2 -7188.038} C_VEL
LIN {X 0,Y 474.726,Z 129.349,A -85,B 0,C 180,E1 -7191.487,E2 -7191.487} C_VEL
LIN {X 0,Y 474.769,Z 129.341,A -85,B 0,C 180,E1 -7194.053,E2 -7194.053} C_VEL
LIN {X 0,Y 474.893,Z 129.328,A -85,B 0,C 180,E1 -7197.456,E2 -7197.456} C_VEL
LIN {X 0,Y 474.91,Z 129.324,A -85,B 0,C 180,E1 -7200,E2 -7200} C_VEL
LIN {X 0,Y 474.893,Z 129.33,A -85,B 0,C 180,E1 -7202.545,E2 -7202.545} C_VEL
LIN {X 0,Y 474.78,Z 129.34,A -85,B 0,C 180,E1 -7205.948,E2 -7205.948} C_VEL
LIN {X 0,Y 474.727,Z 129.352,A -85,B 0,C 180,E1 -7208.514,E2 -7208.514} C_VEL
LIN {X 0,Y 474.703,Z 129.35,A -85,B 0,C 180,E1 -7211.963,E2 -7211.963} C_VEL
LIN {X 0,Y 474.699,Z 129.35,A -85,B 0,C 180,E1 -7215.456,E2 -7215.456} C_VEL
LIN {X 0,Y 474.664,Z 129.356,A -85,B 0,C 180,E1 -7219.011,E2 -7219.011} C_VEL
LIN {X 0,Y 474.587,Z 129.365,A -85,B 0,C 180,E1 -7221.729,E2 -7221.729} C_VEL
LIN {X 0,Y 474.639,Z 129.363,A -85,B 0,C 180,E1 -7224.494,E2 -7224.494} C_VEL
LIN {X 0,Y 474.68,Z 129.352,A -85,B 0,C 180,E1 -7227.335,E2 -7227.335} C_VEL
LIN {X 0,Y 474.605,Z 129.37,A -85,B 0,C 180,E1 -7230.231,E2 -7230.231} C_VEL
LIN {X 0,Y 474.642,Z 129.357,A -85,B 0,C 180,E1 -7233.22,E2 -7233.22} C_VEL
LIN {X 0,Y 474.588,Z 129.369,A -85,B 0,C 180,E1 -7236.324,E2 -7236.324} C_VEL
LIN {X 0,Y 474.649,Z 129.359,A -85,B 0,C 180,E1 -7239.651,E2 -7239.651} C_VEL
LIN {X 0,Y 474.615,Z 129.36,A -85,B 0,C 180,E1 -7242.935,E2 -7242.935} C_VEL
LIN {X 0,Y 474.61,Z 129.369,A -85,B 0,C 180,E1 -7245.896,E2 -7245.896} C_VEL
LIN {X 0,Y 474.628,Z 129.359,A -85,B 0,C 180,E1 -7249.041,E2 -7249.041} C_VEL
LIN {X 0,Y 474.611,Z 129.368,A -85,B 0,C 180,E1 -7251.704,E2 -7251.704} C_VEL
LIN {X 0,Y 474.625,Z 129.359,A -85,B 0,C 180,E1 -7254.726,E2 -7254.726} C_VEL
LIN {X 0,Y 474.637,Z 129.365,A -85,B 0,C 180,E1 -7257.788,E2 -7257.788} C_VEL
LIN {X 0,Y 474.625,Z 129.361,A -85,B 0,C 180,E1 -7260.885,E2 -7260.885} C_VEL
LIN {X 0,Y 474.739,Z 129.427,A -85,B 0,C 180,E1 -7263.248,E2 -7263.248} C_VEL
LIN {X 0,Y 477.043,Z 141.595,A -85,B 0,C 180,E1 -7265.406,E2 -7265.406} C_VEL
LIN {X 0,Y 476.371,Z 159.602,A -85,B 0,C 180,E1 -7268.357,E2 -7268.357} C_VEL
LIN {X 0,Y 475.595,Z 180.319,A -85,B 0,C 180,E1 -7271.699,E2 -7271.699} C_VEL
LIN {X 0,Y 475.233,Z 190.159,A -85,B 0,C 180,E1 -7273.271,E2 -7273.271} C_VEL
LIN {X 0,Y 477.843,Z 209.695,A -85,B 0,C 180,E1 -7273.683,E2 -7273.683} C_VEL
LIN {X 0,Y 477.09,Z 299.277,A -85,B 0,C 180,E1 -7275.143,E2 -7275.143} C_VEL
LIN {X 0,Y 476.713,Z 312.225,A -85,B 0,C 180,E1 -7275.513,E2 -7275.513} C_VEL
LIN {X 0,Y 476.251,Z 325.404,A -85,B 0,C 180,E1 -7276.071,E2 -7276.071} C_VEL
LIN {X 0,Y 475.783,Z 337.341,A -85,B 0,C 180,E1 -7276.765,E2 -7276.765} C_VEL
LIN {X 0,Y 475.34,Z 348.876,A -85,B 0,C 180,E1 -7277.624,E2 -7277.624} C_VEL
LIN {X 0,Y 474.97,Z 359.213,A -85,B 0,C 180,E1 -7278.586,E2 -7278.586} C_VEL
LIN {X 0,Y 474.489,Z 369.344,A -85,B 0,C 180,E1 -7279.762,E2 -7279.762} C_VEL
LIN {X 0,Y 474.19,Z 378.264,A -85,B 0,C 180,E1 -7281.048,E2 -7281.048} C_VEL
LIN {X 0,Y 473.989,Z 385.386,A -85,B 0,C 180,E1 -7282.332,E2 -7282.332} C_VEL
LIN {X 0,Y 473.846,Z 390.958,A -85,B 0,C 180,E1 -7283.585,E2 -7283.585} C_VEL
LIN {X 0,Y 473.831,Z 395.533,A -85,B 0,C 180,E1 -7284.895,E2 -7284.895} C_VEL
LIN {X 0,Y 473.751,Z 397.88,A -85,B 0,C 180,E1 -7285.747,E2 -7285.747} C_VEL
LIN {X 0,Y 473.841,Z 399.797,A -85,B 0,C 180,E1 -7286.599,E2 -7286.599} C_VEL
LIN {X 0,Y 473.793,Z 401.234,A -85,B 0,C 180,E1 -7287.45,E2 -7287.45} C_VEL
LIN {X 0,Y 473.761,Z 402.245,A -85,B 0,C 180,E1 -7288.3,E2 -7288.3} C_VEL
LIN {X 0,Y 473.703,Z 402.855,A -85,B 0,C 180,E1 -7289.15,E2 -7289.15} C_VEL
LIN {X 0,Y 473.693,Z 403.067,A -85,B 0,C 180,E1 -7290,E2 -7290} C_VEL
LIN {X 0,Y 473.703,Z 402.833,A -85,B 0,C 180,E1 -7290.85,E2 -7290.85} C_VEL
LIN {X 0,Y 473.761,Z 402.193,A -85,B 0,C 180,E1 -7291.7,E2 -7291.7} C_VEL
LIN {X 0,Y 473.793,Z 401.151,A -85,B 0,C 180,E1 -7292.551,E2 -7292.551} C_VEL
LIN {X 0,Y 473.842,Z 399.696,A -85,B 0,C 180,E1 -7293.402,E2 -7293.402} C_VEL
LIN {X 0,Y 473.763,Z 396.642,A -85,B 0,C 180,E1 -7294.68,E2 -7294.68} C_VEL
LIN {X 0,Y 473.798,Z 392.523,A -85,B 0,C 180,E1 -7295.96,E2 -7295.96} C_VEL
LIN {X 0,Y 473.972,Z 386.194,A -85,B 0,C 180,E1 -7297.455,E2 -7297.455} C_VEL
LIN {X 0,Y 474.129,Z 379.291,A -85,B 0,C 180,E1 -7298.739,E2 -7298.739} C_VEL
LIN {X 0,Y 474.409,Z 370.728,A -85,B 0,C 180,E1 -7300.025,E2 -7300.025} C_VEL
LIN {X 0,Y 474.786,Z 361.911,A -85,B 0,C 180,E1 -7301.095,E2 -7301.095} C_VEL
LIN {X 0,Y 475.166,Z 351.773,A -85,B 0,C 180,E1 -7302.103,E2 -7302.103} C_VEL
LIN {X 0,Y 475.646,Z 340.324,A -85,B 0,C 180,E1 -7303.023,E2 -7303.023} C_VEL
LIN {X 0,Y 476.165,Z 328.358,A -85,B 0,C 180,E1 -7303.769,E2 -7303.769} C_VEL
LIN {X 0,Y 476.621,Z 315.979,A -85,B 0,C 180,E1 -7304.354,E2 -7304.354} C_VEL
LIN {X 0,Y 476.97,Z 303.402,A -85,B 0,C 180,E1 -7304.779,E2 -7304.779} C_VEL
LIN {X 0,Y 477.233,Z 289.003,A -85,B 0,C 180,E1 -7305.071,E2 -7305.071} C_VEL
LIN {X 0,Y 477.893,Z 208.397,A -85,B 0,C 180,E1 -7306.392,E2 -7306.392} C_VEL
LIN {X 0,Y 475.197,Z 188.549,A -85,B 0,C 180,E1 -7306.847,E2 -7306.847} C_VEL
LIN {X 0,Y 475.75,Z 169.389,A -85,B 0,C 180,E1 -7309.863,E2 -7309.863} C_VEL
LIN {X 0,Y 476.374,Z 151.062,A -85,B 0,C 180,E1 -7312.785,E2 -7312.785} C_VEL
LIN {X 0,Y 476.712,Z 139.738,A -85,B 0,C 180,E1 -7314.613,E2 -7314.613} C_VEL
LIN {X 0,Y 474.711,Z 129.356,A -85,B 0,C 180,E1 -7316.458,E2 -7316.458} C_VEL
LIN {X 0,Y 474.625,Z 129.368,A -85,B 0,C 180,E1 -7319.252,E2 -7319.252} C_VEL
LIN {X 0,Y 474.619,Z 129.369,A -85,B 0,C 180,E1 -7322.431,E2 -7322.431} C_VEL
LIN {X 0,Y 474.618,Z 129.363,A -85,B 0,C 180,E1 -7325.469,E2 -7325.469} C_VEL
LIN {X 0,Y 474.615,Z 129.366,A -85,B 0,C 180,E1 -7328.457,E2 -7328.457} C_VEL
LIN {X 0,Y 474.631,Z 129.361,A -85,B 0,C 180,E1 -7330.959,E2 -7330.959} C_VEL
LIN {X 0,Y 474.613,Z 129.366,A -85,B 0,C 180,E1 -7334.105,E2 -7334.105} C_VEL
LIN {X 0,Y 474.619,Z 129.361,A -85,B 0,C 180,E1 -7337.066,E2 -7337.066} C_VEL
LIN {X 0,Y 474.621,Z 129.359,A -85,B 0,C 180,E1 -7340.354,E2 -7340.354} C_VEL
LIN {X 0,Y 474.592,Z 129.366,A -85,B 0,C 180,E1 -7343.676,E2 -7343.676} C_VEL
LIN {X 0,Y 474.628,Z 129.358,A -85,B 0,C 180,E1 -7346.778,E2 -7346.778} C_VEL
LIN {X 0,Y 474.608,Z 129.366,A -85,B 0,C 180,E1 -7349.77,E2 -7349.77} C_VEL
LIN {X 0,Y 474.701,Z 129.352,A -85,B 0,C 180,E1 -7352.68,E2 -7352.68} C_VEL
LIN {X 0,Y 474.658,Z 129.361,A -85,B 0,C 180,E1 -7355.507,E2 -7355.507} C_VEL
LIN {X 0,Y 474.674,Z 129.358,A -85,B 0,C 180,E1 -7359.185,E2 -7359.185} C_VEL
LIN {X 0,Y 474.647,Z 129.355,A -85,B 0,C 180,E1 -7361.884,E2 -7361.884} C_VEL
LIN {X 0,Y 474.702,Z 129.353,A -85,B 0,C 180,E1 -7364.544,E2 -7364.544} C_VEL
LIN {X 0,Y 474.707,Z 129.351,A -85,B 0,C 180,E1 -7368.037,E2 -7368.037} C_VEL
LIN {X 0,Y 474.714,Z 129.352,A -85,B 0,C 180,E1 -7371.486,E2 -7371.486} C_VEL
LIN {X 0,Y 474.748,Z 129.352,A -85,B 0,C 180,E1 -7374.904,E2 -7374.904} C_VEL
LIN {X 0,Y 474.888,Z 129.331,A -85,B 0,C 180,E1 -7377.455,E2 -7377.455} C_VEL
LIN {X 0,Y 474.912,Z 129.328,A -85,B 0,C 180,E1 -7380,E2 -7380} C_VEL
LIN {X 0,Y 474.884,Z 129.336,A -85,B 0,C 180,E1 -7382.544,E2 -7382.544} C_VEL
LIN {X 0,Y 474.755,Z 129.351,A -85,B 0,C 180,E1 -7385.734,E2 -7385.734} C_VEL
LIN {X 0,Y 475.722,Z 135.461,A -85,B 0,C 180,E1 -7387,E2 -7387} C_VEL
LIN {X 0,Y 475.626,Z 141.837,A -85,B 0,C 180,E1 -7388.249,E2 -7388.249} C_VEL
LIN {X 0,Y 478.348,Z 154.235,A -85,B 0,C 180,E1 -7388.576,E2 -7388.576} C_VEL
LIN {X 0,Y 477.344,Z 248.845,A -85,B 0,C 180,E1 -7390.154,E2 -7390.154} C_VEL
LIN {X 0,Y 477.122,Z 262.441,A -85,B 0,C 180,E1 -7390.556,E2 -7390.556} C_VEL
LIN {X 0,Y 476.81,Z 274.966,A -85,B 0,C 180,E1 -7391.101,E2 -7391.101} C_VEL
LIN {X 0,Y 476.384,Z 287.002,A -85,B 0,C 180,E1 -7391.811,E2 -7391.811} C_VEL
LIN {X 0,Y 475.984,Z 298.516,A -85,B 0,C 180,E1 -7392.687,E2 -7392.687} C_VEL
LIN {X 0,Y 475.534,Z 308.898,A -85,B 0,C 180,E1 -7393.678,E2 -7393.678} C_VEL
LIN {X 0,Y 475.142,Z 318.209,A -85,B 0,C 180,E1 -7394.782,E2 -7394.782} C_VEL
LIN {X 0,Y 474.752,Z 326.681,A -85,B 0,C 180,E1 -7396.018,E2 -7396.018} C_VEL
LIN {X 0,Y 474.446,Z 333.421,A -85,B 0,C 180,E1 -7397.233,E2 -7397.233} C_VEL
LIN {X 0,Y 474.242,Z 339.794,A -85,B 0,C 180,E1 -7398.697,E2 -7398.697} C_VEL
LIN {X 0,Y 474.044,Z 343.988,A -85,B 0,C 180,E1 -7399.937,E2 -7399.937} C_VEL
LIN {X 0,Y 473.931,Z 346.537,A -85,B 0,C 180,E1 -7400.894,E2 -7400.894} C_VEL
LIN {X 0,Y 473.834,Z 348.352,A -85,B 0,C 180,E1 -7401.765,E2 -7401.765} C_VEL
LIN {X 0,Y 473.74,Z 350.27,A -85,B 0,C 180,E1 -7403.106,E2 -7403.106} C_VEL
LIN {X 0,Y 473.69,Z 351.187,A -85,B 0,C 180,E1 -7404.546,E2 -7404.546} C_VEL
LIN {X 0,Y 473.69,Z 351.164,A -85,B 0,C 180,E1 -7405.484,E2 -7405.484} C_VEL
LIN {X 0,Y 473.767,Z 349.972,A -85,B 0,C 180,E1 -7407.119,E2 -7407.119} C_VEL
LIN {X 0,Y 473.812,Z 348.088,A -85,B 0,C 180,E1 -7408.336,E2 -7408.336} C_VEL
LIN {X 0,Y 473.981,Z 344.699,A -85,B 0,C 180,E1 -7409.783,E2 -7409.783} C_VEL
LIN {X 0,Y 474.069,Z 339.851,A -85,B 0,C 180,E1 -7411.256,E2 -7411.256} C_VEL
LIN {X 0,Y 474.392,Z 333.493,A -85,B 0,C 180,E1 -7412.718,E2 -7412.718} C_VEL
LIN {X 0,Y 474.644,Z 326.504,A -85,B 0,C 180,E1 -7413.985,E2 -7413.985} C_VEL
LIN {X 0,Y 475.02,Z 317.854,A -85,B 0,C 180,E1 -7415.24,E2 -7415.24} C_VEL
LIN {X 0,Y 475.416,Z 308.157,A -85,B 0,C 180,E1 -7416.381,E2 -7416.381} C_VEL
LIN {X 0,Y 475.863,Z 297.322,A -85,B 0,C 180,E1 -7417.399,E2 -7417.399} C_VEL
LIN {X 0,Y 476.272,Z 285.255,A -85,B 0,C 180,E1 -7418.298,E2 -7418.298} C_VEL
LIN {X 0,Y 476.668,Z 273.368,A -85,B 0,C 180,E1 -7418.98,E2 -7418.98} C_VEL
LIN {X 0,Y 476.93,Z 260.191,A -85,B 0,C 180,E1 -7419.535,E2 -7419.535} C_VEL
LIN {X 0,Y 477.183,Z 248.026,A -85,B 0,C 180,E1 -7419.881,E2 -7419.881} C_VEL
LIN {X 0,Y 478.034,Z 158.659,A -85,B 0,C 180,E1 -7421.338,E2 -7421.338} C_VEL
LIN {X 0,Y 477.317,Z 156.755,A -85,B 0,C 180,E1 -7421.394,E2 -7421.394} C_VEL
LIN {X 0,Y 474.501,Z 154.531,A -85,B 0,C 180,E1 -7421.528,E2 -7421.528} C_VEL
LIN {X 0,Y 471.164,Z 152.101,A -85,B 0,C 180,E1 -7421.683,E2 -7421.683} C_VEL
LIN {X 0,Y 470.338,Z 150.488,A -85,B 0,C 180,E1 -7421.739,E2 -7421.739} C_VEL
LIN {X 0,Y 468.449,Z 140.989,A -85,B 0,C 180,E1 -7421.973,E2 -7421.973} C_VEL
LIN {X 0,Y 468.428,Z 134.922,A -85,B 0,C 180,E1 -7423.258,E2 -7423.258} C_VEL
LIN {X 0,Y 467.663,Z 130.232,A -85,B 0,C 180,E1 -7424.321,E2 -7424.321} C_VEL
LIN {X 0,Y 467.589,Z 130.242,A -85,B 0,C 180,E1 -7427.44,E2 -7427.44} C_VEL
